LIN {X -0.212,Y -660.705,Z 1253.356,A 0.000,B 0.000,C 90.000,E1 100.141} C_DIS
LIN {X 0.232,Y -659.495,Z 1253.354,A 0.000,B 0.000,C 90.000,E1 99.613} C_DIS
LIN {X 0.124,Y -658.795,Z 1253.352,A 0.000,B 0.000,C 90.000,E1 99.378} C_DIS
LIN {X -0.205,Y -657.112,Z 1253.349,A 0.000,B 0.000,C 90.000,E1 98.916} C_DIS
LIN {X 0.108,Y -655.018,Z 1253.347,A 0.000,B 0.000,C 90.000,E1 98.398} C_DIS
LIN {X -0.260,Y -651.900,Z 1253.343,A 0.000,B 0.000,C 90.000,E1 97.814} C_DIS
LIN {X 0.015,Y -649.059,Z 1253.341,A 0.000,B 0.000,C 90.000,E1 97.296} C_DIS
LIN {X 0.153,Y -644.946,Z 1253.337,A 0.000,B 0.000,C 90.000,E1 96.663} C_DIS
LIN {X 0.258,Y -640.230,Z 1253.334,A 0.000,B 0.000,C 90.000,E1 96.030} C_DIS
LIN {X -0.052,Y -637.232,Z 1253.332,A 0.000,B 0.000,C 90.000,E1 95.682} C_DIS
LIN {X -0.011,Y -631.428,Z 1253.328,A 0.000,B 0.000,C 90.000,E1 95.049} C_DIS
LIN {X 0.272,Y -626.430,Z 1253.325,A 0.000,B 0.000,C 90.000,E1 94.531} C_DIS
LIN {X 0.030,Y -619.785,Z 1253.322,A 0.000,B 0.000,C 90.000,E1 93.955} C_DIS
LIN {X 0.104,Y -612.877,Z 1253.319,A 0.000,B 0.000,C 90.000,E1 93.383} C_DIS
LIN {X 0.178,Y -610.033,Z 1253.318,A 0.000,B 0.000,C 90.000,E1 93.154} C_DIS
LIN {X 0.140,Y -602.473,Z 1253.315,A 0.000,B 0.000,C 90.000,E1 92.636} C_DIS
LIN {X 0.166,Y -596.282,Z 1253.313,A 0.000,B 0.000,C 90.000,E1 92.236} C_DIS
LIN {X -0.229,Y -589.784,Z 1253.310,A 0.000,B 0.000,C 90.000,E1 91.892} C_DIS
LIN {X -0.265,Y -582.813,Z 1253.308,A 0.000,B 0.000,C 90.000,E1 91.547} C_DIS
LIN {X 0.065,Y -571.892,Z 1253.306,A 0.000,B 0.000,C 90.000,E1 91.088} C_DIS
LIN {X -0.005,Y -570.760,Z 1253.306,A 0.000,B 0.000,C 90.000,E1 91.031} C_DIS
LIN {X -0.074,Y -568.415,Z 1253.305,A 0.000,B 0.000,C 90.000,E1 90.859} C_DIS
LIN {X -0.108,Y -568.400,Z 1253.305,A 0.000,B 0.000,C 90.000,E1 90.859} C_DIS
LIN {X -0.110,Y -567.219,Z 1253.303,A 0.000,B 0.000,C 90.000,E1 90.516} C_DIS
LIN {X 0.015,Y -567.116,Z 1253.300,A 0.000,B 0.000,C 90.000,E1 90.057} C_DIS
LIN {X 0.207,Y -568.765,Z 1253.287,A 0.000,B 0.000,C 90.000,E1 87.707} C_DIS
LIN {X 0.001,Y -570.383,Z 1253.277,A 0.000,B 0.000,C 90.000,E1 85.812} C_DIS
LIN {X 0.269,Y -572.026,Z 1253.268,A 0.000,B 0.000,C 90.000,E1 84.147} C_DIS
LIN {X -0.071,Y -573.481,Z 1253.260,A 0.000,B 0.000,C 90.000,E1 82.818} C_DIS
LIN {X 0.021,Y -575.454,Z 1253.250,A 0.000,B 0.000,C 90.000,E1 80.905} C_DIS
LIN {X 0.191,Y -576.493,Z 1253.244,A 0.000,B 0.000,C 90.000,E1 79.803} C_DIS
LIN {X 0.012,Y -577.547,Z 1253.236,A 0.000,B 0.000,C 90.000,E1 78.465} C_DIS
LIN {X -0.254,Y -578.363,Z 1253.230,A 0.000,B 0.000,C 90.000,E1 77.409} C_DIS
LIN {X 0.065,Y -579.449,Z 1253.221,A 0.000,B 0.000,C 90.000,E1 75.755} C_DIS
LIN {X 0.188,Y -580.267,Z 1253.214,A 0.000,B 0.000,C 90.000,E1 74.393} C_DIS
LIN {X -0.241,Y -581.061,Z 1253.206,A 0.000,B 0.000,C 90.000,E1 73.087} C_DIS
LIN {X 0.106,Y -582.211,Z 1253.195,A 0.000,B 0.000,C 90.000,E1 71.167} C_DIS
LIN {X -0.144,Y -582.836,Z 1253.189,A 0.000,B 0.000,C 90.000,E1 70.115} C_DIS
LIN {X -0.251,Y -584.179,Z 1253.178,A 0.000,B 0.000,C 90.000,E1 67.975} C_DIS
LIN {X -0.130,Y -586.270,Z 1253.163,A 0.000,B 0.000,C 90.000,E1 65.281} C_DIS
LIN {X 0.004,Y -588.112,Z 1253.151,A 0.000,B 0.000,C 90.000,E1 63.127} C_DIS
LIN {X 0.091,Y -590.450,Z 1253.137,A 0.000,B 0.000,C 90.000,E1 60.717} C_DIS
LIN {X -0.152,Y -591.819,Z 1253.130,A 0.000,B 0.000,C 90.000,E1 59.410} C_DIS
LIN {X 0.030,Y -592.949,Z 1253.124,A 0.000,B 0.000,C 90.000,E1 58.329} C_DIS
LIN {X 0.120,Y -594.284,Z 1253.117,A 0.000,B 0.000,C 90.000,E1 56.993} C_DIS
LIN {X 0.277,Y -595.738,Z 1253.108,A 0.000,B 0.000,C 90.000,E1 55.388} C_DIS
LIN {X -0.244,Y -596.930,Z 1253.101,A 0.000,B 0.000,C 90.000,E1 54.116} C_DIS
LIN {X 0.326,Y -598.249,Z 1253.092,A 0.000,B 0.000,C 90.000,E1 52.477} C_DIS
LIN {X 0.204,Y -599.273,Z 1253.084,A 0.000,B 0.000,C 90.000,E1 51.170} C_DIS
LIN {X -0.149,Y -599.925,Z 1253.079,A 0.000,B 0.000,C 90.000,E1 50.150} C_DIS
LIN {X -0.307,Y -600.765,Z 1253.068,A 0.000,B 0.000,C 90.000,E1 48.324} C_DIS
LIN {X -0.064,Y -601.171,Z 1253.061,A 0.000,B 0.000,C 90.000,E1 46.986} C_DIS
LIN {X 0.188,Y -601.494,Z 1253.054,A 0.000,B 0.000,C 90.000,E1 45.648} C_DIS
LIN {X 0.217,Y -601.534,Z 1253.048,A 0.000,B 0.000,C 90.000,E1 44.595} C_DIS
LIN {X 0.244,Y -601.354,Z 1253.042,A 0.000,B 0.000,C 90.000,E1 43.542} C_DIS
LIN {X -0.148,Y -601.034,Z 1253.036,A 0.000,B 0.000,C 90.000,E1 42.528} C_DIS
LIN {X -0.069,Y -600.444,Z 1253.027,A 0.000,B 0.000,C 90.000,E1 40.943} C_DIS
LIN {X -0.019,Y -599.846,Z 1253.022,A 0.000,B 0.000,C 90.000,E1 39.886} C_DIS
LIN {X 0.258,Y -599.022,Z 1253.014,A 0.000,B 0.000,C 90.000,E1 38.543} C_DIS
LIN {X -0.334,Y -598.349,Z 1253.010,A 0.000,B 0.000,C 90.000,E1 37.810} C_DIS
LIN {X 0.136,Y -597.246,Z 1253.004,A 0.000,B 0.000,C 90.000,E1 36.710} C_DIS
LIN {X -0.119,Y -595.857,Z 1252.998,A 0.000,B 0.000,C 90.000,E1 35.678} C_DIS
LIN {X -0.149,Y -595.087,Z 1252.995,A 0.000,B 0.000,C 90.000,E1 35.152} C_DIS
LIN {X 0.064,Y -593.240,Z 1252.989,A 0.000,B 0.000,C 90.000,E1 34.072} C_DIS
LIN {X 0.090,Y -591.042,Z 1252.984,A 0.000,B 0.000,C 90.000,E1 33.007} C_DIS
LIN {X 0.056,Y -589.056,Z 1252.979,A 0.000,B 0.000,C 90.000,E1 32.212} C_DIS
LIN {X 0.010,Y -586.738,Z 1252.975,A 0.000,B 0.000,C 90.000,E1 31.416} C_DIS
LIN {X 0.243,Y -584.098,Z 1252.970,A 0.000,B 0.000,C 90.000,E1 30.590} C_DIS
LIN {X 0.143,Y -580.969,Z 1252.966,A 0.000,B 0.000,C 90.000,E1 29.795} C_DIS
LIN {X -0.130,Y -578.685,Z 1252.963,A 0.000,B 0.000,C 90.000,E1 29.283} C_DIS
LIN {X -0.133,Y -576.179,Z 1252.960,A 0.000,B 0.000,C 90.000,E1 28.743} C_DIS
LIN {X 0.069,Y -573.479,Z 1252.957,A 0.000,B 0.000,C 90.000,E1 28.180} C_DIS
LIN {X 0.019,Y -570.606,Z 1252.954,A 0.000,B 0.000,C 90.000,E1 27.641} C_DIS
LIN {X 0.100,Y -566.694,Z 1252.950,A 0.000,B 0.000,C 90.000,E1 26.950} C_DIS
LIN {X -0.007,Y -563.312,Z 1252.947,A 0.000,B 0.000,C 90.000,E1 26.411} C_DIS
LIN {X -0.088,Y -557.862,Z 1252.942,A 0.000,B 0.000,C 90.000,E1 25.591} C_DIS
LIN {X -0.112,Y -552.822,Z 1252.938,A 0.000,B 0.000,C 90.000,E1 24.899} C_DIS
LIN {X -0.222,Y -546.312,Z 1252.934,A 0.000,B 0.000,C 90.000,E1 24.079} C_DIS
LIN {X 0.149,Y -540.407,Z 1252.930,A 0.000,B 0.000,C 90.000,E1 23.334} C_DIS
LIN {X 0.178,Y -533.117,Z 1252.925,A 0.000,B 0.000,C 90.000,E1 22.514} C_DIS
LIN {X -0.235,Y -525.243,Z 1252.921,A 0.000,B 0.000,C 90.000,E1 21.716} C_DIS
LIN {X 0.015,Y -516.052,Z 1252.915,A 0.000,B 0.000,C 90.000,E1 20.737} C_DIS
LIN {X -0.065,Y -505.488,Z 1252.909,A 0.000,B 0.000,C 90.000,E1 19.685} C_DIS
LIN {X 0.052,Y -495.616,Z 1252.904,A 0.000,B 0.000,C 90.000,E1 18.725} C_DIS
LIN {X -0.104,Y -486.934,Z 1252.900,A 0.000,B 0.000,C 90.000,E1 17.946} C_DIS
LIN {X -0.065,Y -478.380,Z 1252.895,A 0.000,B 0.000,C 90.000,E1 17.166} C_DIS
LIN {X -0.049,Y -462.047,Z 1252.887,A 0.000,B 0.000,C 90.000,E1 15.717} C_DIS
LIN {X -0.194,Y -444.342,Z 1252.878,A 0.000,B 0.000,C 90.000,E1 14.120} C_DIS
LIN {X -0.038,Y -421.556,Z 1252.866,A 0.000,B 0.000,C 90.000,E1 11.827} C_DIS
LIN {X 0.078,Y -407.325,Z 1252.857,A 0.000,B 0.000,C 90.000,E1 10.254} C_DIS
LIN {X 0.105,Y -401.563,Z 1252.854,A 0.000,B 0.000,C 90.000,E1 9.613} C_DIS
LIN {X 0.063,Y -397.092,Z 1252.850,A 0.000,B 0.000,C 90.000,E1 9.029} C_DIS
LIN {X 0.041,Y -395.063,Z 1252.848,A 0.000,B 0.000,C 90.000,E1 8.681} C_DIS
LIN {X 0.176,Y -394.571,Z 1252.848,A 0.000,B 0.000,C 90.000,E1 8.568} C_DIS
LIN {X 0.138,Y -394.543,Z 1252.848,A 0.000,B 0.000,C 90.000,E1 8.568} C_DIS
LIN {X 0.073,Y -394.451,Z 1252.847,A 0.000,B 0.000,C 90.000,E1 8.511} C_DIS
LIN {X 0.035,Y -394.445,Z 1252.847,A 0.000,B 0.000,C 90.000,E1 8.511} C_DIS
LIN {X 0.137,Y -396.450,Z 1252.845,A 0.000,B 0.000,C 90.000,E1 8.049} C_DIS
LIN {X -0.191,Y -399.766,Z 1252.843,A 0.000,B 0.000,C 90.000,E1 7.757} C_DIS
LIN {X 0.059,Y -403.844,Z 1252.841,A 0.000,B 0.000,C 90.000,E1 7.409} C_DIS
LIN {X -0.125,Y -413.483,Z 1252.838,A 0.000,B 0.000,C 90.000,E1 6.777} C_DIS
LIN {X -0.006,Y -423.027,Z 1252.834,A 0.000,B 0.000,C 90.000,E1 6.087} C_DIS
LIN {X -0.107,Y -430.941,Z 1252.831,A 0.000,B 0.000,C 90.000,E1 5.511} C_DIS
LIN {X 0.128,Y -438.553,Z 1252.827,A 0.000,B 0.000,C 90.000,E1 4.878} C_DIS
LIN {X -0.106,Y -452.599,Z 1252.821,A 0.000,B 0.000,C 90.000,E1 3.784} C_DIS
LIN {X -0.122,Y -460.203,Z 1252.818,A 0.000,B 0.000,C 90.000,E1 3.154} C_DIS
LIN {X 0.232,Y -467.575,Z 1252.814,A 0.000,B 0.000,C 90.000,E1 2.465} C_DIS
LIN {X 0.122,Y -473.346,Z 1252.811,A 0.000,B 0.000,C 90.000,E1 1.949} C_DIS
LIN {X -0.172,Y -478.953,Z 1252.808,A 0.000,B 0.000,C 90.000,E1 1.432} C_DIS
LIN {X 0.010,Y -485.708,Z 1252.804,A 0.000,B 0.000,C 90.000,E1 0.688} C_DIS
LIN {X 0.000,Y -491.571,Z 1252.800,A 0.000,B 0.000,C 90.000,E1 360.000} C_DIS
LIN {X 0.034,Y -495.782,Z 1252.797,A 0.000,B 0.000,C 90.000,E1 359.484} C_DIS
LIN {X -0.059,Y -501.360,Z 1252.793,A 0.000,B 0.000,C 90.000,E1 358.740} C_DIS
LIN {X -0.089,Y -506.541,Z 1252.789,A 0.000,B 0.000,C 90.000,E1 357.993} C_DIS
LIN {X -0.087,Y -511.392,Z 1252.785,A 0.000,B 0.000,C 90.000,E1 357.249} C_DIS
LIN {X 0.202,Y -516.817,Z 1252.780,A 0.000,B 0.000,C 90.000,E1 356.331} C_DIS
LIN {X -0.129,Y -519.389,Z 1252.777,A 0.000,B 0.000,C 90.000,E1 355.927} C_DIS
LIN {X 0.022,Y -523.280,Z 1252.773,A 0.000,B 0.000,C 90.000,E1 355.179} C_DIS
LIN {X 0.207,Y -526.904,Z 1252.769,A 0.000,B 0.000,C 90.000,E1 354.432} C_DIS
LIN {X 0.180,Y -529.625,Z 1252.766,A 0.000,B 0.000,C 90.000,E1 353.856} C_DIS
LIN {X 0.171,Y -532.171,Z 1252.763,A 0.000,B 0.000,C 90.000,E1 353.280} C_DIS
LIN {X 0.221,Y -535.546,Z 1252.758,A 0.000,B 0.000,C 90.000,E1 352.413} C_DIS
LIN {X -0.229,Y -538.689,Z 1252.753,A 0.000,B 0.000,C 90.000,E1 351.602} C_DIS
LIN {X -0.114,Y -541.618,Z 1252.749,A 0.000,B 0.000,C 90.000,E1 350.735} C_DIS
LIN {X 0.122,Y -544.158,Z 1252.744,A 0.000,B 0.000,C 90.000,E1 349.859} C_DIS
LIN {X -0.155,Y -547.318,Z 1252.738,A 0.000,B 0.000,C 90.000,E1 348.757} C_DIS
LIN {X -0.287,Y -550.077,Z 1252.731,A 0.000,B 0.000,C 90.000,E1 347.645} C_DIS
LIN {X -0.140,Y -553.217,Z 1252.724,A 0.000,B 0.000,C 90.000,E1 346.228} C_DIS
LIN {X -0.320,Y -554.809,Z 1252.719,A 0.000,B 0.000,C 90.000,E1 345.408} C_DIS
LIN {X -0.221,Y -556.749,Z 1252.713,A 0.000,B 0.000,C 90.000,E1 344.283} C_DIS
LIN {X 0.060,Y -558.427,Z 1252.706,A 0.000,B 0.000,C 90.000,E1 343.142} C_DIS
LIN {X -0.163,Y -559.792,Z 1252.700,A 0.000,B 0.000,C 90.000,E1 342.054} C_DIS
LIN {X 0.167,Y -560.813,Z 1252.694,A 0.000,B 0.000,C 90.000,E1 340.913} C_DIS
LIN {X -0.026,Y -561.387,Z 1252.688,A 0.000,B 0.000,C 90.000,E1 339.826} C_DIS
LIN {X -0.336,Y -561.509,Z 1252.683,A 0.000,B 0.000,C 90.000,E1 339.028} C_DIS
LIN {X 0.085,Y -561.263,Z 1252.679,A 0.000,B 0.000,C 90.000,E1 338.156} C_DIS
LIN {X -0.224,Y -560.706,Z 1252.674,A 0.000,B 0.000,C 90.000,E1 337.358} C_DIS
LIN {X 0.192,Y -559.841,Z 1252.670,A 0.000,B 0.000,C 90.000,E1 336.485} C_DIS
LIN {X 0.087,Y -558.671,Z 1252.665,A 0.000,B 0.000,C 90.000,E1 335.665} C_DIS
LIN {X -0.029,Y -557.185,Z 1252.660,A 0.000,B 0.000,C 90.000,E1 334.845} C_DIS
LIN {X 0.122,Y -554.796,Z 1252.654,A 0.000,B 0.000,C 90.000,E1 333.717} C_DIS
LIN {X -0.095,Y -554.002,Z 1252.653,A 0.000,B 0.000,C 90.000,E1 333.461} C_DIS
LIN {X -0.065,Y -553.388,Z 1252.651,A 0.000,B 0.000,C 90.000,E1 333.179} C_DIS
LIN {X -0.243,Y -550.785,Z 1252.646,A 0.000,B 0.000,C 90.000,E1 332.359} C_DIS
LIN {X -0.195,Y -547.731,Z 1252.642,A 0.000,B 0.000,C 90.000,E1 331.513} C_DIS
LIN {X 0.187,Y -546.009,Z 1252.639,A 0.000,B 0.000,C 90.000,E1 331.051} C_DIS
LIN {X -0.169,Y -542.745,Z 1252.635,A 0.000,B 0.000,C 90.000,E1 330.383} C_DIS
LIN {X -0.082,Y -539.018,Z 1252.631,A 0.000,B 0.000,C 90.000,E1 329.665} C_DIS
LIN {X 0.106,Y -535.654,Z 1252.628,A 0.000,B 0.000,C 90.000,E1 329.076} C_DIS
LIN {X 0.221,Y -528.187,Z 1252.622,A 0.000,B 0.000,C 90.000,E1 327.916} C_DIS
LIN {X 0.040,Y -520.383,Z 1252.616,A 0.000,B 0.000,C 90.000,E1 326.786} C_DIS
LIN {X 0.033,Y -515.805,Z 1252.612,A 0.000,B 0.000,C 90.000,E1 326.087} C_DIS
LIN {X -0.050,Y -512.575,Z 1252.609,A 0.000,B 0.000,C 90.000,E1 325.548} C_DIS
LIN {X -0.109,Y -509.785,Z 1252.606,A 0.000,B 0.000,C 90.000,E1 325.022} C_DIS
LIN {X 0.129,Y -507.435,Z 1252.602,A 0.000,B 0.000,C 90.000,E1 324.402} C_DIS
LIN {X -0.024,Y -505.761,Z 1252.599,A 0.000,B 0.000,C 90.000,E1 323.829} C_DIS
LIN {X 0.180,Y -504.597,Z 1252.596,A 0.000,B 0.000,C 90.000,E1 323.210} C_DIS
LIN {X -0.034,Y -503.754,Z 1252.592,A 0.000,B 0.000,C 90.000,E1 322.637} C_DIS
LIN {X -0.056,Y -503.268,Z 1252.588,A 0.000,B 0.000,C 90.000,E1 321.743} C_DIS
LIN {X -0.012,Y -503.780,Z 1252.569,A 0.000,B 0.000,C 90.000,E1 318.447} C_DIS
LIN {X -0.210,Y -504.378,Z 1252.558,A 0.000,B 0.000,C 90.000,E1 316.377} C_DIS
LIN {X 0.195,Y -504.702,Z 1252.549,A 0.000,B 0.000,C 90.000,E1 314.838} C_DIS
LIN {X -0.109,Y -505.060,Z 1252.541,A 0.000,B 0.000,C 90.000,E1 313.380} C_DIS
LIN {X 0.057,Y -505.627,Z 1252.529,A 0.000,B 0.000,C 90.000,E1 311.272} C_DIS
LIN {X 0.060,Y -505.992,Z 1252.519,A 0.000,B 0.000,C 90.000,E1 309.483} C_DIS
LIN {X 0.056,Y -506.474,Z 1252.508,A 0.000,B 0.000,C 90.000,E1 307.397} C_DIS
LIN {X -0.040,Y -506.824,Z 1252.501,A 0.000,B 0.000,C 90.000,E1 306.217} C_DIS
LIN {X -0.029,Y -507.013,Z 1252.495,A 0.000,B 0.000,C 90.000,E1 305.025} C_DIS
LIN {X 0.302,Y -507.136,Z 1252.486,A 0.000,B 0.000,C 90.000,E1 303.499} C_DIS
LIN {X -0.018,Y -507.187,Z 1252.476,A 0.000,B 0.000,C 90.000,E1 301.750} C_DIS
LIN {X 0.149,Y -507.117,Z 1252.470,A 0.000,B 0.000,C 90.000,E1 300.541} C_DIS
LIN {X 0.261,Y -507.099,Z 1252.460,A 0.000,B 0.000,C 90.000,E1 298.743} C_DIS
LIN {X -0.122,Y -506.892,Z 1252.450,A 0.000,B 0.000,C 90.000,E1 297.001} C_DIS
LIN {X 0.127,Y -506.793,Z 1252.437,A 0.000,B 0.000,C 90.000,E1 294.591} C_DIS
LIN {X 0.246,Y -506.796,Z 1252.430,A 0.000,B 0.000,C 90.000,E1 293.387} C_DIS
LIN {X 0.253,Y -506.480,Z 1252.422,A 0.000,B 0.000,C 90.000,E1 291.897} C_DIS
LIN {X 0.158,Y -505.684,Z 1252.412,A 0.000,B 0.000,C 90.000,E1 290.120} C_DIS
LIN {X -0.113,Y -504.623,Z 1252.399,A 0.000,B 0.000,C 90.000,E1 287.764} C_DIS
LIN {X 0.051,Y -504.205,Z 1252.392,A 0.000,B 0.000,C 90.000,E1 286.551} C_DIS
LIN {X -0.014,Y -503.519,Z 1252.384,A 0.000,B 0.000,C 90.000,E1 285.064} C_DIS
LIN {X -0.217,Y -502.611,Z 1252.375,A 0.000,B 0.000,C 90.000,E1 283.592} C_DIS
LIN {X 0.054,Y -501.572,Z 1252.367,A 0.000,B 0.000,C 90.000,E1 282.063} C_DIS
LIN {X 0.202,Y -500.426,Z 1252.359,A 0.000,B 0.000,C 90.000,E1 280.546} C_DIS
LIN {X 0.170,Y -499.181,Z 1252.349,A 0.000,B 0.000,C 90.000,E1 278.746} C_DIS
LIN {X 0.103,Y -498.052,Z 1252.339,A 0.000,B 0.000,C 90.000,E1 276.947} C_DIS
LIN {X 0.138,Y -496.782,Z 1252.325,A 0.000,B 0.000,C 90.000,E1 274.531} C_DIS
LIN {X 0.106,Y -496.101,Z 1252.319,A 0.000,B 0.000,C 90.000,E1 273.326} C_DIS
LIN {X -0.070,Y -495.051,Z 1252.310,A 0.000,B 0.000,C 90.000,E1 271.835} C_DIS
LIN {X -0.210,Y -493.235,Z 1252.297,A 0.000,B 0.000,C 90.000,E1 269.427} C_DIS
LIN {X -0.046,Y -491.472,Z 1252.281,A 0.000,B 0.000,C 90.000,E1 266.674} C_DIS
LIN {X 0.048,Y -490.478,Z 1252.271,A 0.000,B 0.000,C 90.000,E1 264.837} C_DIS
LIN {X -0.161,Y -489.520,Z 1252.263,A 0.000,B 0.000,C 90.000,E1 263.337} C_DIS
LIN {X -0.269,Y -488.598,Z 1252.256,A 0.000,B 0.000,C 90.000,E1 262.129} C_DIS
LIN {X 0.108,Y -487.122,Z 1252.248,A 0.000,B 0.000,C 90.000,E1 260.557} C_DIS
LIN {X -0.027,Y -484.754,Z 1252.232,A 0.000,B 0.000,C 90.000,E1 257.813} C_DIS
LIN {X -0.086,Y -483.773,Z 1252.224,A 0.000,B 0.000,C 90.000,E1 256.284} C_DIS
LIN {X 0.128,Y -482.296,Z 1252.210,A 0.000,B 0.000,C 90.000,E1 253.795} C_DIS
LIN {X 0.108,Y -481.096,Z 1252.198,A 0.000,B 0.000,C 90.000,E1 251.638} C_DIS
LIN {X -0.083,Y -480.146,Z 1252.188,A 0.000,B 0.000,C 90.000,E1 249.806} C_DIS
LIN {X 0.158,Y -479.290,Z 1252.179,A 0.000,B 0.000,C 90.000,E1 248.230} C_DIS
LIN {X 0.275,Y -478.309,Z 1252.169,A 0.000,B 0.000,C 90.000,E1 246.357} C_DIS
LIN {X -0.046,Y -477.192,Z 1252.160,A 0.000,B 0.000,C 90.000,E1 244.845} C_DIS
LIN {X 0.063,Y -476.372,Z 1252.153,A 0.000,B 0.000,C 90.000,E1 243.589} C_DIS
LIN {X 0.127,Y -475.332,Z 1252.145,A 0.000,B 0.000,C 90.000,E1 242.025} C_DIS
LIN {X 0.175,Y -474.196,Z 1252.136,A 0.000,B 0.000,C 90.000,E1 240.461} C_DIS
LIN {X 0.028,Y -472.895,Z 1252.127,A 0.000,B 0.000,C 90.000,E1 238.918} C_DIS
LIN {X 0.030,Y -471.234,Z 1252.117,A 0.000,B 0.000,C 90.000,E1 237.041} C_DIS
LIN {X 0.004,Y -469.467,Z 1252.105,A 0.000,B 0.000,C 90.000,E1 234.848} C_DIS
LIN {X -0.093,Y -467.634,Z 1252.089,A 0.000,B 0.000,C 90.000,E1 232.029} C_DIS
LIN {X 0.047,Y -466.757,Z 1252.080,A 0.000,B 0.000,C 90.000,E1 230.436} C_DIS
LIN {X 0.102,Y -465.962,Z 1252.072,A 0.000,B 0.000,C 90.000,E1 228.852} C_DIS
LIN {X -0.208,Y -464.988,Z 1252.063,A 0.000,B 0.000,C 90.000,E1 227.310} C_DIS
LIN {X -0.019,Y -464.409,Z 1252.057,A 0.000,B 0.000,C 90.000,E1 226.338} C_DIS
LIN {X 0.075,Y -463.196,Z 1252.045,A 0.000,B 0.000,C 90.000,E1 224.109} C_DIS
LIN {X 0.105,Y -463.920,Z 1252.001,A 0.000,B 0.000,C 90.000,E1 216.171} C_DIS
LIN {X -0.204,Y -467.553,Z 1251.975,A 0.000,B 0.000,C 90.000,E1 211.465} C_DIS
LIN {X -0.065,Y -469.195,Z 1251.966,A 0.000,B 0.000,C 90.000,E1 209.873} C_DIS
LIN {X 0.047,Y -471.564,Z 1251.955,A 0.000,B 0.000,C 90.000,E1 207.975} C_DIS
LIN {X 0.120,Y -474.587,Z 1251.942,A 0.000,B 0.000,C 90.000,E1 205.463} C_DIS
LIN {X 0.153,Y -477.199,Z 1251.931,A 0.000,B 0.000,C 90.000,E1 203.590} C_DIS
LIN {X -0.192,Y -480.139,Z 1251.921,A 0.000,B 0.000,C 90.000,E1 201.770} C_DIS
LIN {X -0.198,Y -487.630,Z 1251.899,A 0.000,B 0.000,C 90.000,E1 197.764} C_DIS
LIN {X -0.032,Y -492.178,Z 1251.887,A 0.000,B 0.000,C 90.000,E1 195.607} C_DIS
LIN {X 0.086,Y -496.168,Z 1251.877,A 0.000,B 0.000,C 90.000,E1 193.772} C_DIS
LIN {X 0.104,Y -500.904,Z 1251.865,A 0.000,B 0.000,C 90.000,E1 191.658} C_DIS
LIN {X 0.205,Y -505.202,Z 1251.855,A 0.000,B 0.000,C 90.000,E1 189.849} C_DIS
LIN {X -0.142,Y -508.773,Z 1251.847,A 0.000,B 0.000,C 90.000,E1 188.398} C_DIS
LIN {X 0.073,Y -512.473,Z 1251.838,A 0.000,B 0.000,C 90.000,E1 186.891} C_DIS
LIN {X 0.208,Y -516.783,Z 1251.828,A 0.000,B 0.000,C 90.000,E1 185.106} C_DIS
LIN {X -0.118,Y -521.062,Z 1251.819,A 0.000,B 0.000,C 90.000,E1 183.383} C_DIS
LIN {X -0.248,Y -523.131,Z 1251.814,A 0.000,B 0.000,C 90.000,E1 182.522} C_DIS
LIN {X 0.058,Y -527.258,Z 1251.804,A 0.000,B 0.000,C 90.000,E1 180.745} C_DIS
LIN {X -0.097,Y -531.938,Z 1251.793,A 0.000,B 0.000,C 90.000,E1 178.740} C_DIS
LIN {X -0.127,Y -535.076,Z 1251.785,A 0.000,B 0.000,C 90.000,E1 177.306} C_DIS
LIN {X -0.105,Y -537.453,Z 1251.779,A 0.000,B 0.000,C 90.000,E1 176.159} C_DIS
LIN {X -0.010,Y -539.672,Z 1251.772,A 0.000,B 0.000,C 90.000,E1 175.008} C_DIS
LIN {X 0.125,Y -541.805,Z 1251.766,A 0.000,B 0.000,C 90.000,E1 173.856} C_DIS
LIN {X -0.173,Y -544.326,Z 1251.758,A 0.000,B 0.000,C 90.000,E1 172.470} C_DIS
LIN {X 0.107,Y -546.651,Z 1251.750,A 0.000,B 0.000,C 90.000,E1 171.027} C_DIS
LIN {X -0.143,Y -547.931,Z 1251.746,A 0.000,B 0.000,C 90.000,E1 170.208} C_DIS
LIN {X -0.150,Y -550.380,Z 1251.736,A 0.000,B 0.000,C 90.000,E1 168.522} C_DIS
LIN {X -0.125,Y -552.219,Z 1251.728,A 0.000,B 0.000,C 90.000,E1 167.117} C_DIS
LIN {X -0.240,Y -554.690,Z 1251.718,A 0.000,B 0.000,C 90.000,E1 165.172} C_DIS
LIN {X 0.127,Y -557.921,Z 1251.705,A 0.000,B 0.000,C 90.000,E1 162.906} C_DIS
LIN {X 0.201,Y -560.782,Z 1251.697,A 0.000,B 0.000,C 90.000,E1 161.511} C_DIS
LIN {X 0.146,Y -564.530,Z 1251.690,A 0.000,B 0.000,C 90.000,E1 160.134} C_DIS
LIN {X -0.134,Y -567.235,Z 1251.685,A 0.000,B 0.000,C 90.000,E1 159.337} C_DIS
LIN {X 0.226,Y -573.289,Z 1251.677,A 0.000,B 0.000,C 90.000,E1 157.794} C_DIS
LIN {X -0.268,Y -579.586,Z 1251.669,A 0.000,B 0.000,C 90.000,E1 156.485} C_DIS
LIN {X -0.116,Y -589.402,Z 1251.659,A 0.000,B 0.000,C 90.000,E1 154.588} C_DIS
LIN {X -0.042,Y -595.848,Z 1251.652,A 0.000,B 0.000,C 90.000,E1 153.384} C_DIS
LIN {X 0.125,Y -602.111,Z 1251.646,A 0.000,B 0.000,C 90.000,E1 152.180} C_DIS
LIN {X 0.158,Y -607.430,Z 1251.640,A 0.000,B 0.000,C 90.000,E1 151.129} C_DIS
LIN {X -0.284,Y -613.138,Z 1251.633,A 0.000,B 0.000,C 90.000,E1 149.999} C_DIS
LIN {X -0.100,Y -618.079,Z 1251.627,A 0.000,B 0.000,C 90.000,E1 148.948} C_DIS
LIN {X -0.057,Y -622.984,Z 1251.622,A 0.000,B 0.000,C 90.000,E1 147.916} C_DIS
LIN {X 0.251,Y -626.523,Z 1251.618,A 0.000,B 0.000,C 90.000,E1 147.120} C_DIS
LIN {X -0.112,Y -630.963,Z 1251.612,A 0.000,B 0.000,C 90.000,E1 146.135} C_DIS
LIN {X 0.112,Y -635.093,Z 1251.606,A 0.000,B 0.000,C 90.000,E1 145.102} C_DIS
LIN {X -0.133,Y -638.991,Z 1251.601,A 0.000,B 0.000,C 90.000,E1 144.116} C_DIS
LIN {X -0.331,Y -642.466,Z 1251.595,A 0.000,B 0.000,C 90.000,E1 143.130} C_DIS
LIN {X -0.005,Y -644.870,Z 1251.591,A 0.000,B 0.000,C 90.000,E1 142.351} C_DIS
LIN {X -0.164,Y -647.119,Z 1251.587,A 0.000,B 0.000,C 90.000,E1 141.618} C_DIS
LIN {X 0.128,Y -649.963,Z 1251.581,A 0.000,B 0.000,C 90.000,E1 140.598} C_DIS
LIN {X -0.044,Y -652.657,Z 1251.576,A 0.000,B 0.000,C 90.000,E1 139.622} C_DIS
LIN {X -0.228,Y -655.941,Z 1251.569,A 0.000,B 0.000,C 90.000,E1 138.405} C_DIS
LIN {X 0.084,Y -659.085,Z 1251.562,A 0.000,B 0.000,C 90.000,E1 137.148} C_DIS
LIN {X -0.066,Y -664.648,Z 1251.550,A 0.000,B 0.000,C 90.000,E1 134.960} C_DIS
LIN {X -0.064,Y -669.295,Z 1251.540,A 0.000,B 0.000,C 90.000,E1 133.257} C_DIS
LIN {X -0.454,Y -673.284,Z 1251.532,A 0.000,B 0.000,C 90.000,E1 131.838} C_DIS
LIN {X -0.299,Y -676.540,Z 1251.526,A 0.000,B 0.000,C 90.000,E1 130.620} C_DIS
LIN {X 0.027,Y -680.306,Z 1251.518,A 0.000,B 0.000,C 90.000,E1 129.152} C_DIS
LIN {X -0.135,Y -683.438,Z 1251.511,A 0.000,B 0.000,C 90.000,E1 127.971} C_DIS
LIN {X 0.324,Y -687.147,Z 1251.503,A 0.000,B 0.000,C 90.000,E1 126.503} C_DIS
LIN {X -0.200,Y -689.408,Z 1251.498,A 0.000,B 0.000,C 90.000,E1 125.598} C_DIS
LIN {X -0.091,Y -692.088,Z 1251.491,A 0.000,B 0.000,C 90.000,E1 124.405} C_DIS
LIN {X 0.024,Y -694.104,Z 1251.486,A 0.000,B 0.000,C 90.000,E1 123.452} C_DIS
LIN {X -0.153,Y -696.980,Z 1251.478,A 0.000,B 0.000,C 90.000,E1 122.054} C_DIS
LIN {X -0.091,Y -699.143,Z 1251.472,A 0.000,B 0.000,C 90.000,E1 120.875} C_DIS
LIN {X 0.373,Y -701.187,Z 1251.465,A 0.000,B 0.000,C 90.000,E1 119.667} C_DIS
LIN {X 0.238,Y -702.592,Z 1251.460,A 0.000,B 0.000,C 90.000,E1 118.743} C_DIS
LIN {X -0.214,Y -703.742,Z 1251.455,A 0.000,B 0.000,C 90.000,E1 117.847} C_DIS
LIN {X 0.302,Y -704.627,Z 1251.449,A 0.000,B 0.000,C 90.000,E1 116.873} C_DIS
LIN {X 0.222,Y -704.991,Z 1251.446,A 0.000,B 0.000,C 90.000,E1 116.181} C_DIS
LIN {X 0.167,Y -705.110,Z 1251.443,A 0.000,B 0.000,C 90.000,E1 115.720} C_DIS
LIN {X 0.093,Y -704.864,Z 1251.439,A 0.000,B 0.000,C 90.000,E1 115.027} C_DIS
LIN {X -0.265,Y -704.481,Z 1251.437,A 0.000,B 0.000,C 90.000,E1 114.591} C_DIS
LIN {X 0.305,Y -703.686,Z 1251.434,A 0.000,B 0.000,C 90.000,E1 114.079} C_DIS
LIN {X -0.341,Y -703.002,Z 1251.433,A 0.000,B 0.000,C 90.000,E1 113.898} C_DIS
LIN {X 0.217,Y -700.978,Z 1251.430,A 0.000,B 0.000,C 90.000,E1 113.387} C_DIS
LIN {X 0.353,Y -700.259,Z 1251.429,A 0.000,B 0.000,C 90.000,E1 113.259} C_DIS
LIN {X -0.035,Y -696.034,Z 1251.427,A 0.000,B 0.000,C 90.000,E1 112.823} C_DIS
LIN {X 0.093,Y -694.744,Z 1251.426,A 0.000,B 0.000,C 90.000,E1 112.695} C_DIS
LIN {X 0.010,Y -692.786,Z 1251.426,A 0.000,B 0.000,C 90.000,E1 112.589} C_DIS
LIN {X 0.094,Y -687.962,Z 1251.425,A 0.000,B 0.000,C 90.000,E1 112.408} C_DIS
LIN {X 0.256,Y -685.952,Z 1251.424,A 0.000,B 0.000,C 90.000,E1 112.333} C_DIS
LIN {X -0.193,Y -677.441,Z 1251.424,A 0.000,B 0.000,C 90.000,E1 112.259} C_DIS
LIN {X 0.393,Y -676.916,Z 1251.424,A 0.000,B 0.000,C 90.000,E1 112.206} C_DIS
LIN {X 0.327,Y -627.513,Z 1251.424,A 0.000,B 0.000,C 90.000,E1 112.206} C_DIS
LIN {X -0.031,Y -626.466,Z 1251.423,A 0.000,B 0.000,C 90.000,E1 112.206} C_DIS
LIN {X -0.088,Y -625.366,Z 1251.423,A 0.000,B 0.000,C 90.000,E1 112.153} C_DIS
LIN {X -0.240,Y -623.489,Z 1251.422,A 0.000,B 0.000,C 90.000,E1 112.025} C_DIS
LIN {X -0.276,Y -623.476,Z 1251.422,A 0.000,B 0.000,C 90.000,E1 112.025} C_DIS
LIN {X -0.104,Y -623.241,Z 1251.422,A 0.000,B 0.000,C 90.000,E1 111.897} C_DIS
LIN {X 0.096,Y -624.519,Z 1251.419,A 0.000,B 0.000,C 90.000,E1 111.482} C_DIS
LIN {X 0.092,Y -627.194,Z 1251.417,A 0.000,B 0.000,C 90.000,E1 110.972} C_DIS
LIN {X -0.076,Y -632.344,Z 1251.412,A 0.000,B 0.000,C 90.000,E1 110.120} C_DIS
LIN {X -0.374,Y -636.282,Z 1251.408,A 0.000,B 0.000,C 90.000,E1 109.396} C_DIS
LIN {X -0.241,Y -642.292,Z 1251.401,A 0.000,B 0.000,C 90.000,E1 108.127} C_DIS
LIN {X -0.151,Y -649.418,Z 1251.392,A 0.000,B 0.000,C 90.000,E1 106.622} C_DIS
LIN {X 0.253,Y -652.682,Z 1251.388,A 0.000,B 0.000,C 90.000,E1 105.843} C_DIS
LIN {X 0.004,Y -654.638,Z 1251.385,A 0.000,B 0.000,C 90.000,E1 105.371} C_DIS
LIN {X -0.179,Y -657.121,Z 1251.381,A 0.000,B 0.000,C 90.000,E1 104.647} C_DIS
LIN {X 0.237,Y -658.503,Z 1251.379,A 0.000,B 0.000,C 90.000,E1 104.120} C_DIS
LIN {X -0.078,Y -659.996,Z 1251.375,A 0.000,B 0.000,C 90.000,E1 103.411} C_DIS
LIN {X 0.362,Y -660.734,Z 1251.372,A 0.000,B 0.000,C 90.000,E1 102.883} C_DIS
LIN {X 0.164,Y -661.217,Z 1251.369,A 0.000,B 0.000,C 90.000,E1 102.411} C_DIS
LIN {X -0.171,Y -661.335,Z 1251.366,A 0.000,B 0.000,C 90.000,E1 101.951} C_DIS
LIN {X -0.267,Y -661.311,Z 1251.365,A 0.000,B 0.000,C 90.000,E1 101.715} C_DIS
LIN {X 0.185,Y -660.980,Z 1251.362,A 0.000,B 0.000,C 90.000,E1 101.186} C_DIS
LIN {X -0.016,Y -660.411,Z 1251.360,A 0.000,B 0.000,C 90.000,E1 100.715} C_DIS
LIN {X 0.307,Y -659.531,Z 1251.357,A 0.000,B 0.000,C 90.000,E1 100.197} C_DIS
LIN {X 0.092,Y -658.371,Z 1251.354,A 0.000,B 0.000,C 90.000,E1 99.726} C_DIS
LIN {X -0.129,Y -657.735,Z 1251.353,A 0.000,B 0.000,C 90.000,E1 99.500} C_DIS
LIN {X 0.289,Y -656.043,Z 1251.350,A 0.000,B 0.000,C 90.000,E1 98.973} C_DIS
LIN {X -0.054,Y -653.991,Z 1251.347,A 0.000,B 0.000,C 90.000,E1 98.511} C_DIS
LIN {X 0.214,Y -650.930,Z 1251.344,A 0.000,B 0.000,C 90.000,E1 97.871} C_DIS
LIN {X -0.279,Y -647.352,Z 1251.340,A 0.000,B 0.000,C 90.000,E1 97.296} C_DIS
LIN {X -0.034,Y -644.064,Z 1251.338,A 0.000,B 0.000,C 90.000,E1 96.777} C_DIS
LIN {X 0.063,Y -639.397,Z 1251.334,A 0.000,B 0.000,C 90.000,E1 96.144} C_DIS
LIN {X 0.297,Y -635.316,Z 1251.331,A 0.000,B 0.000,C 90.000,E1 95.625} C_DIS
LIN {X -0.130,Y -630.685,Z 1251.329,A 0.000,B 0.000,C 90.000,E1 95.163} C_DIS
LIN {X 0.163,Y -624.448,Z 1251.325,A 0.000,B 0.000,C 90.000,E1 94.531} C_DIS
LIN {X -0.067,Y -617.714,Z 1251.322,A 0.000,B 0.000,C 90.000,E1 93.955} C_DIS
LIN {X -0.020,Y -610.651,Z 1251.319,A 0.000,B 0.000,C 90.000,E1 93.383} C_DIS
LIN {X -0.239,Y -604.655,Z 1251.317,A 0.000,B 0.000,C 90.000,E1 92.980} C_DIS
LIN {X -0.082,Y -597.007,Z 1251.314,A 0.000,B 0.000,C 90.000,E1 92.465} C_DIS
LIN {X -0.261,Y -588.955,Z 1251.311,A 0.000,B 0.000,C 90.000,E1 92.007} C_DIS
LIN {X -0.247,Y -581.992,Z 1251.309,A 0.000,B 0.000,C 90.000,E1 91.661} C_DIS
LIN {X 0.166,Y -571.236,Z 1251.307,A 0.000,B 0.000,C 90.000,E1 91.203} C_DIS
LIN {X 0.062,Y -570.056,Z 1251.306,A 0.000,B 0.000,C 90.000,E1 91.146} C_DIS
LIN {X 0.167,Y -567.933,Z 1251.306,A 0.000,B 0.000,C 90.000,E1 90.974} C_DIS
LIN {X 0.132,Y -567.903,Z 1251.306,A 0.000,B 0.000,C 90.000,E1 90.974} C_DIS
LIN {X 0.030,Y -567.764,Z 1251.305,A 0.000,B 0.000,C 90.000,E1 90.859} C_DIS
LIN {X 0.041,Y -566.945,Z 1251.303,A 0.000,B 0.000,C 90.000,E1 90.516} C_DIS
LIN {X -0.174,Y -567.007,Z 1251.300,A 0.000,B 0.000,C 90.000,E1 90.057} C_DIS
LIN {X -0.024,Y -568.202,Z 1251.291,A 0.000,B 0.000,C 90.000,E1 88.396} C_DIS
LIN {X -0.254,Y -569.747,Z 1251.281,A 0.000,B 0.000,C 90.000,E1 86.502} C_DIS
LIN {X -0.271,Y -571.840,Z 1251.268,A 0.000,B 0.000,C 90.000,E1 84.318} C_DIS
LIN {X -0.042,Y -573.280,Z 1251.261,A 0.000,B 0.000,C 90.000,E1 82.932} C_DIS
LIN {X -0.040,Y -575.238,Z 1251.250,A 0.000,B 0.000,C 90.000,E1 81.027} C_DIS
LIN {X 0.118,Y -576.264,Z 1251.244,A 0.000,B 0.000,C 90.000,E1 79.926} C_DIS
LIN {X -0.171,Y -577.147,Z 1251.238,A 0.000,B 0.000,C 90.000,E1 78.870} C_DIS
LIN {X -0.222,Y -578.131,Z 1251.231,A 0.000,B 0.000,C 90.000,E1 77.521} C_DIS
LIN {X 0.086,Y -578.878,Z 1251.225,A 0.000,B 0.000,C 90.000,E1 76.408} C_DIS
LIN {X 0.197,Y -579.754,Z 1251.217,A 0.000,B 0.000,C 90.000,E1 75.046} C_DIS
LIN {X -0.023,Y -580.706,Z 1251.208,A 0.000,B 0.000,C 90.000,E1 73.449} C_DIS
LIN {X -0.237,Y -581.782,Z 1251.198,A 0.000,B 0.000,C 90.000,E1 71.583} C_DIS
LIN {X 0.260,Y -582.606,Z 1251.190,A 0.000,B 0.000,C 90.000,E1 70.188} C_DIS
LIN {X 0.135,Y -583.951,Z 1251.178,A 0.000,B 0.000,C 90.000,E1 68.050} C_DIS
LIN {X 0.235,Y -586.038,Z 1251.163,A 0.000,B 0.000,C 90.000,E1 65.357} C_DIS
LIN {X -0.172,Y -587.877,Z 1251.151,A 0.000,B 0.000,C 90.000,E1 63.256} C_DIS
LIN {X -0.091,Y -590.208,Z 1251.138,A 0.000,B 0.000,C 90.000,E1 60.845} C_DIS
LIN {X -0.337,Y -591.576,Z 1251.131,A 0.000,B 0.000,C 90.000,E1 59.537} C_DIS
LIN {X -0.265,Y -592.982,Z 1251.123,A 0.000,B 0.000,C 90.000,E1 58.201} C_DIS
LIN {X -0.068,Y -594.078,Z 1251.117,A 0.000,B 0.000,C 90.000,E1 57.120} C_DIS
LIN {X 0.088,Y -595.499,Z 1251.109,A 0.000,B 0.000,C 90.000,E1 55.515} C_DIS
LIN {X 0.051,Y -596.704,Z 1251.101,A 0.000,B 0.000,C 90.000,E1 54.196} C_DIS
LIN {X 0.010,Y -598.247,Z 1251.091,A 0.000,B 0.000,C 90.000,E1 52.351} C_DIS
LIN {X 0.018,Y -599.047,Z 1251.085,A 0.000,B 0.000,C 90.000,E1 51.295} C_DIS
LIN {X 0.128,Y -599.725,Z 1251.079,A 0.000,B 0.000,C 90.000,E1 50.231} C_DIS
LIN {X -0.056,Y -600.299,Z 1251.072,A 0.000,B 0.000,C 90.000,E1 48.933} C_DIS
LIN {X -0.248,Y -600.634,Z 1251.068,A 0.000,B 0.000,C 90.000,E1 48.162} C_DIS
LIN {X 0.411,Y -600.974,Z 1251.063,A 0.000,B 0.000,C 90.000,E1 47.310} C_DIS
LIN {X 0.031,Y -601.273,Z 1251.054,A 0.000,B 0.000,C 90.000,E1 45.769} C_DIS
LIN {X 0.050,Y -601.384,Z 1251.048,A 0.000,B 0.000,C 90.000,E1 44.717} C_DIS
LIN {X -0.348,Y -601.210,Z 1251.043,A 0.000,B 0.000,C 90.000,E1 43.704} C_DIS
LIN {X 0.317,Y -600.990,Z 1251.038,A 0.000,B 0.000,C 90.000,E1 42.852} C_DIS
LIN {X -0.290,Y -600.520,Z 1251.031,A 0.000,B 0.000,C 90.000,E1 41.595} C_DIS
LIN {X -0.245,Y -600.031,Z 1251.025,A 0.000,B 0.000,C 90.000,E1 40.539} C_DIS
LIN {X 0.014,Y -599.562,Z 1251.021,A 0.000,B 0.000,C 90.000,E1 39.725} C_DIS
LIN {X 0.044,Y -598.938,Z 1251.015,A 0.000,B 0.000,C 90.000,E1 38.669} C_DIS
LIN {X -0.081,Y -598.280,Z 1251.010,A 0.000,B 0.000,C 90.000,E1 37.890} C_DIS
LIN {X -0.211,Y -596.862,Z 1251.003,A 0.000,B 0.000,C 90.000,E1 36.583} C_DIS
LIN {X -0.120,Y -595.421,Z 1250.997,A 0.000,B 0.000,C 90.000,E1 35.518} C_DIS
LIN {X -0.011,Y -594.591,Z 1250.994,A 0.000,B 0.000,C 90.000,E1 34.978} C_DIS
LIN {X 0.044,Y -592.719,Z 1250.989,A 0.000,B 0.000,C 90.000,E1 33.913} C_DIS
LIN {X -0.265,Y -590.415,Z 1250.983,A 0.000,B 0.000,C 90.000,E1 32.880} C_DIS
LIN {X -0.182,Y -589.100,Z 1250.980,A 0.000,B 0.000,C 90.000,E1 32.339} C_DIS
LIN {X -0.109,Y -587.619,Z 1250.977,A 0.000,B 0.000,C 90.000,E1 31.799} C_DIS
LIN {X -0.170,Y -585.090,Z 1250.972,A 0.000,B 0.000,C 90.000,E1 31.003} C_DIS
LIN {X 0.004,Y -584.225,Z 1250.971,A 0.000,B 0.000,C 90.000,E1 30.718} C_DIS
LIN {X -0.094,Y -581.114,Z 1250.966,A 0.000,B 0.000,C 90.000,E1 29.922} C_DIS
LIN {X 0.281,Y -577.676,Z 1250.962,A 0.000,B 0.000,C 90.000,E1 29.077} C_DIS
LIN {X -0.087,Y -574.434,Z 1250.958,A 0.000,B 0.000,C 90.000,E1 28.437} C_DIS
LIN {X 0.212,Y -570.100,Z 1250.953,A 0.000,B 0.000,C 90.000,E1 27.590} C_DIS
LIN {X -0.126,Y -566.989,Z 1250.950,A 0.000,B 0.000,C 90.000,E1 27.078} C_DIS
LIN {X 0.275,Y -563.661,Z 1250.947,A 0.000,B 0.000,C 90.000,E1 26.488} C_DIS
LIN {X -0.204,Y -559.168,Z 1250.943,A 0.000,B 0.000,C 90.000,E1 25.848} C_DIS
LIN {X -0.006,Y -556.305,Z 1250.941,A 0.000,B 0.000,C 90.000,E1 25.412} C_DIS
LIN {X -0.322,Y -553.292,Z 1250.939,A 0.000,B 0.000,C 90.000,E1 25.027} C_DIS
LIN {X -0.045,Y -545.682,Z 1250.933,A 0.000,B 0.000,C 90.000,E1 24.027} C_DIS
LIN {X -0.173,Y -539.722,Z 1250.930,A 0.000,B 0.000,C 90.000,E1 23.334} C_DIS
LIN {X 0.019,Y -534.919,Z 1250.927,A 0.000,B 0.000,C 90.000,E1 22.770} C_DIS
LIN {X 0.207,Y -525.836,Z 1250.921,A 0.000,B 0.000,C 90.000,E1 21.770} C_DIS
LIN {X -0.076,Y -516.610,Z 1250.916,A 0.000,B 0.000,C 90.000,E1 20.844} C_DIS
LIN {X -0.007,Y -505.894,Z 1250.910,A 0.000,B 0.000,C 90.000,E1 19.758} C_DIS
LIN {X 0.190,Y -495.853,Z 1250.905,A 0.000,B 0.000,C 90.000,E1 18.779} C_DIS
LIN {X -0.019,Y -487.161,Z 1250.900,A 0.000,B 0.000,C 90.000,E1 18.000} C_DIS
LIN {X 0.028,Y -480.008,Z 1250.896,A 0.000,B 0.000,C 90.000,E1 17.347} C_DIS
LIN {X -0.018,Y -471.087,Z 1250.892,A 0.000,B 0.000,C 90.000,E1 16.567} C_DIS
LIN {X 0.216,Y -459.286,Z 1250.886,A 0.000,B 0.000,C 90.000,E1 15.481} C_DIS
LIN {X -0.086,Y -437.220,Z 1250.875,A 0.000,B 0.000,C 90.000,E1 13.467} C_DIS
LIN {X 0.130,Y -417.054,Z 1250.863,A 0.000,B 0.000,C 90.000,E1 11.366} C_DIS
LIN {X -0.125,Y -405.588,Z 1250.856,A 0.000,B 0.000,C 90.000,E1 10.141} C_DIS
LIN {X -0.155,Y -401.308,Z 1250.854,A 0.000,B 0.000,C 90.000,E1 9.670} C_DIS
LIN {X -0.159,Y -397.023,Z 1250.850,A 0.000,B 0.000,C 90.000,E1 9.095} C_DIS
LIN {X -0.134,Y -394.507,Z 1250.848,A 0.000,B 0.000,C 90.000,E1 8.624} C_DIS
LIN {X -0.172,Y -394.485,Z 1250.848,A 0.000,B 0.000,C 90.000,E1 8.624} C_DIS
LIN {X 0.191,Y -394.399,Z 1250.848,A 0.000,B 0.000,C 90.000,E1 8.511} C_DIS
LIN {X 0.153,Y -394.403,Z 1250.847,A 0.000,B 0.000,C 90.000,E1 8.511} C_DIS
LIN {X -0.022,Y -396.303,Z 1250.845,A 0.000,B 0.000,C 90.000,E1 8.106} C_DIS
LIN {X 0.023,Y -399.519,Z 1250.843,A 0.000,B 0.000,C 90.000,E1 7.757} C_DIS
LIN {X 0.150,Y -401.201,Z 1250.842,A 0.000,B 0.000,C 90.000,E1 7.587} C_DIS
LIN {X -0.093,Y -410.073,Z 1250.839,A 0.000,B 0.000,C 90.000,E1 7.004} C_DIS
LIN {X -0.002,Y -419.754,Z 1250.835,A 0.000,B 0.000,C 90.000,E1 6.315} C_DIS
LIN {X -0.126,Y -429.417,Z 1250.831,A 0.000,B 0.000,C 90.000,E1 5.625} C_DIS
LIN {X 0.002,Y -438.653,Z 1250.827,A 0.000,B 0.000,C 90.000,E1 4.878} C_DIS
LIN {X -0.110,Y -452.535,Z 1250.821,A 0.000,B 0.000,C 90.000,E1 3.784} C_DIS
LIN {X -0.160,Y -461.580,Z 1250.817,A 0.000,B 0.000,C 90.000,E1 3.037} C_DIS
LIN {X -0.166,Y -467.549,Z 1250.814,A 0.000,B 0.000,C 90.000,E1 2.522} C_DIS
LIN {X -0.243,Y -473.311,Z 1250.811,A 0.000,B 0.000,C 90.000,E1 2.007} C_DIS
LIN {X 0.196,Y -478.682,Z 1250.808,A 0.000,B 0.000,C 90.000,E1 1.432} C_DIS
LIN {X 0.032,Y -485.366,Z 1250.804,A 0.000,B 0.000,C 90.000,E1 0.745} C_DIS
LIN {X 0.000,Y -491.800,Z 1250.800,A 0.000,B 0.000,C 90.000,E1 360.000} C_DIS
LIN {X 0.035,Y -496.035,Z 1250.797,A 0.000,B 0.000,C 90.000,E1 359.484} C_DIS
LIN {X 0.132,Y -502.717,Z 1250.792,A 0.000,B 0.000,C 90.000,E1 358.568} C_DIS
LIN {X -0.083,Y -506.888,Z 1250.789,A 0.000,B 0.000,C 90.000,E1 357.993} C_DIS
LIN {X -0.077,Y -511.741,Z 1250.785,A 0.000,B 0.000,C 90.000,E1 357.249} C_DIS
LIN {X -0.005,Y -516.323,Z 1250.781,A 0.000,B 0.000,C 90.000,E1 356.502} C_DIS
LIN {X -0.112,Y -519.769,Z 1250.777,A 0.000,B 0.000,C 90.000,E1 355.927} C_DIS
LIN {X 0.042,Y -523.692,Z 1250.773,A 0.000,B 0.000,C 90.000,E1 355.179} C_DIS
LIN {X 0.231,Y -527.317,Z 1250.769,A 0.000,B 0.000,C 90.000,E1 354.432} C_DIS
LIN {X 0.208,Y -530.036,Z 1250.766,A 0.000,B 0.000,C 90.000,E1 353.856} C_DIS
LIN {X 0.203,Y -532.581,Z 1250.763,A 0.000,B 0.000,C 90.000,E1 353.280} C_DIS
LIN {X 0.257,Y -535.987,Z 1250.758,A 0.000,B 0.000,C 90.000,E1 352.413} C_DIS
LIN {X -0.187,Y -539.097,Z 1250.753,A 0.000,B 0.000,C 90.000,E1 351.602} C_DIS
LIN {X -0.068,Y -542.025,Z 1250.749,A 0.000,B 0.000,C 90.000,E1 350.735} C_DIS
LIN {X 0.173,Y -544.564,Z 1250.744,A 0.000,B 0.000,C 90.000,E1 349.859} C_DIS
LIN {X -0.097,Y -547.736,Z 1250.738,A 0.000,B 0.000,C 90.000,E1 348.757} C_DIS
LIN {X -0.224,Y -550.511,Z 1250.731,A 0.000,B 0.000,C 90.000,E1 347.645} C_DIS
LIN {X -0.068,Y -553.621,Z 1250.724,A 0.000,B 0.000,C 90.000,E1 346.228} C_DIS
LIN {X -0.244,Y -555.270,Z 1250.719,A 0.000,B 0.000,C 90.000,E1 345.408} C_DIS
LIN {X 0.141,Y -557.662,Z 1250.711,A 0.000,B 0.000,C 90.000,E1 343.976} C_DIS
LIN {X -0.256,Y -559.263,Z 1250.705,A 0.000,B 0.000,C 90.000,E1 342.906} C_DIS
LIN {X -0.065,Y -560.305,Z 1250.700,A 0.000,B 0.000,C 90.000,E1 342.054} C_DIS
LIN {X 0.272,Y -561.346,Z 1250.694,A 0.000,B 0.000,C 90.000,E1 340.913} C_DIS
LIN {X -0.036,Y -561.858,Z 1250.690,A 0.000,B 0.000,C 90.000,E1 340.115} C_DIS
LIN {X 0.191,Y -562.096,Z 1250.685,A 0.000,B 0.000,C 90.000,E1 339.263} C_DIS
LIN {X 0.099,Y -562.146,Z 1250.682,A 0.000,B 0.000,C 90.000,E1 338.720} C_DIS
LIN {X -0.204,Y -561.843,Z 1250.677,A 0.000,B 0.000,C 90.000,E1 337.922} C_DIS
LIN {X 0.223,Y -561.197,Z 1250.673,A 0.000,B 0.000,C 90.000,E1 337.050} C_DIS
LIN {X 0.130,Y -560.290,Z 1250.668,A 0.000,B 0.000,C 90.000,E1 336.230} C_DIS
LIN {X 0.235,Y -559.483,Z 1250.665,A 0.000,B 0.000,C 90.000,E1 335.665} C_DIS
LIN {X 0.128,Y -558.030,Z 1250.660,A 0.000,B 0.000,C 90.000,E1 334.845} C_DIS
LIN {X -0.207,Y -555.656,Z 1250.654,A 0.000,B 0.000,C 90.000,E1 333.768} C_DIS
LIN {X -0.141,Y -554.373,Z 1250.651,A 0.000,B 0.000,C 90.000,E1 333.204} C_DIS
LIN {X 0.164,Y -552.561,Z 1250.648,A 0.000,B 0.000,C 90.000,E1 332.615} C_DIS
LIN {X -0.059,Y -551.791,Z 1250.646,A 0.000,B 0.000,C 90.000,E1 332.359} C_DIS
LIN {X -0.003,Y -548.733,Z 1250.642,A 0.000,B 0.000,C 90.000,E1 331.513} C_DIS
LIN {X 0.265,Y -546.432,Z 1250.639,A 0.000,B 0.000,C 90.000,E1 330.923} C_DIS
LIN {X -0.088,Y -543.086,Z 1250.635,A 0.000,B 0.000,C 90.000,E1 330.255} C_DIS
LIN {X 0.000,Y -539.327,Z 1250.631,A 0.000,B 0.000,C 90.000,E1 329.537} C_DIS
LIN {X 0.046,Y -534.918,Z 1250.627,A 0.000,B 0.000,C 90.000,E1 328.820} C_DIS
LIN {X 0.304,Y -528.358,Z 1250.621,A 0.000,B 0.000,C 90.000,E1 327.788} C_DIS
LIN {X -0.243,Y -521.327,Z 1250.616,A 0.000,B 0.000,C 90.000,E1 326.834} C_DIS
LIN {X -0.086,Y -516.440,Z 1250.612,A 0.000,B 0.000,C 90.000,E1 326.087} C_DIS
LIN {X 0.146,Y -513.119,Z 1250.609,A 0.000,B 0.000,C 90.000,E1 325.515} C_DIS
LIN {X -0.301,Y -509.922,Z 1250.605,A 0.000,B 0.000,C 90.000,E1 324.975} C_DIS
LIN {X -0.017,Y -507.618,Z 1250.602,A 0.000,B 0.000,C 90.000,E1 324.356} C_DIS
LIN {X -0.177,Y -505.961,Z 1250.599,A 0.000,B 0.000,C 90.000,E1 323.783} C_DIS
LIN {X 0.250,Y -504.354,Z 1250.594,A 0.000,B 0.000,C 90.000,E1 322.844} C_DIS
LIN {X -0.074,Y -503.629,Z 1250.589,A 0.000,B 0.000,C 90.000,E1 321.984} C_DIS
LIN {X -0.147,Y -504.191,Z 1250.569,A 0.000,B 0.000,C 90.000,E1 318.405} C_DIS
LIN {X 0.001,Y -504.801,Z 1250.557,A 0.000,B 0.000,C 90.000,E1 316.296} C_DIS
LIN {X 0.189,Y -505.078,Z 1250.551,A 0.000,B 0.000,C 90.000,E1 315.081} C_DIS
LIN {X 0.119,Y -505.506,Z 1250.541,A 0.000,B 0.000,C 90.000,E1 313.299} C_DIS
LIN {X -0.037,Y -506.102,Z 1250.529,A 0.000,B 0.000,C 90.000,E1 311.229} C_DIS
LIN {X -0.014,Y -506.510,Z 1250.519,A 0.000,B 0.000,C 90.000,E1 309.439} C_DIS
LIN {X -0.087,Y -507.006,Z 1250.508,A 0.000,B 0.000,C 90.000,E1 307.363} C_DIS
LIN {X -0.075,Y -507.339,Z 1250.501,A 0.000,B 0.000,C 90.000,E1 306.171} C_DIS
LIN {X -0.050,Y -507.523,Z 1250.494,A 0.000,B 0.000,C 90.000,E1 304.978} C_DIS
LIN {X 0.198,Y -507.697,Z 1250.484,A 0.000,B 0.000,C 90.000,E1 303.166} C_DIS
LIN {X 0.159,Y -507.760,Z 1250.474,A 0.000,B 0.000,C 90.000,E1 301.386} C_DIS
LIN {X -0.089,Y -507.701,Z 1250.463,A 0.000,B 0.000,C 90.000,E1 299.333} C_DIS
LIN {X -0.176,Y -507.610,Z 1250.456,A 0.000,B 0.000,C 90.000,E1 298.153} C_DIS
LIN {X 0.268,Y -507.454,Z 1250.448,A 0.000,B 0.000,C 90.000,E1 296.616} C_DIS
LIN {X -0.236,Y -507.436,Z 1250.437,A 0.000,B 0.000,C 90.000,E1 294.591} C_DIS
LIN {X -0.203,Y -507.457,Z 1250.432,A 0.000,B 0.000,C 90.000,E1 293.695} C_DIS
LIN {X -0.087,Y -507.121,Z 1250.422,A 0.000,B 0.000,C 90.000,E1 291.897} C_DIS
LIN {X -0.167,Y -506.339,Z 1250.412,A 0.000,B 0.000,C 90.000,E1 290.120} C_DIS
LIN {X 0.147,Y -505.190,Z 1250.397,A 0.000,B 0.000,C 90.000,E1 287.402} C_DIS
LIN {X 0.239,Y -504.876,Z 1250.392,A 0.000,B 0.000,C 90.000,E1 286.496} C_DIS
LIN {X 0.190,Y -504.192,Z 1250.384,A 0.000,B 0.000,C 90.000,E1 285.009} C_DIS
LIN {X 0.002,Y -503.274,Z 1250.375,A 0.000,B 0.000,C 90.000,E1 283.536} C_DIS
LIN {X -0.202,Y -502.232,Z 1250.367,A 0.000,B 0.000,C 90.000,E1 282.063} C_DIS
LIN {X -0.041,Y -501.115,Z 1250.359,A 0.000,B 0.000,C 90.000,E1 280.546} C_DIS
LIN {X -0.057,Y -499.901,Z 1250.349,A 0.000,B 0.000,C 90.000,E1 278.746} C_DIS
LIN {X -0.252,Y -498.588,Z 1250.337,A 0.000,B 0.000,C 90.000,E1 276.663} C_DIS
LIN {X -0.050,Y -497.594,Z 1250.325,A 0.000,B 0.000,C 90.000,E1 274.531} C_DIS
LIN {X -0.069,Y -496.902,Z 1250.318,A 0.000,B 0.000,C 90.000,E1 273.326} C_DIS
LIN {X -0.214,Y -495.826,Z 1250.310,A 0.000,B 0.000,C 90.000,E1 271.833} C_DIS
LIN {X 0.004,Y -493.745,Z 1250.295,A 0.000,B 0.000,C 90.000,E1 269.083} C_DIS
LIN {X -0.222,Y -492.645,Z 1250.286,A 0.000,B 0.000,C 90.000,E1 267.593} C_DIS
LIN {X -0.158,Y -492.154,Z 1250.281,A 0.000,B 0.000,C 90.000,E1 266.674} C_DIS
LIN {X -0.049,Y -491.174,Z 1250.271,A 0.000,B 0.000,C 90.000,E1 264.837} C_DIS
LIN {X 0.040,Y -490.623,Z 1250.266,A 0.000,B 0.000,C 90.000,E1 263.913} C_DIS
LIN {X -0.161,Y -489.530,Z 1250.258,A 0.000,B 0.000,C 90.000,E1 262.413} C_DIS
LIN {X 0.162,Y -488.107,Z 1250.249,A 0.000,B 0.000,C 90.000,E1 260.849} C_DIS
LIN {X -0.063,Y -485.433,Z 1250.232,A 0.000,B 0.000,C 90.000,E1 257.813} C_DIS
LIN {X 0.230,Y -484.243,Z 1250.222,A 0.000,B 0.000,C 90.000,E1 255.936} C_DIS
LIN {X 0.124,Y -482.981,Z 1250.210,A 0.000,B 0.000,C 90.000,E1 253.795} C_DIS
LIN {X 0.122,Y -481.741,Z 1250.198,A 0.000,B 0.000,C 90.000,E1 251.638} C_DIS
LIN {X -0.056,Y -480.803,Z 1250.188,A 0.000,B 0.000,C 90.000,E1 249.806} C_DIS
LIN {X -0.247,Y -479.997,Z 1250.179,A 0.000,B 0.000,C 90.000,E1 248.284} C_DIS
LIN {X -0.109,Y -478.939,Z 1250.169,A 0.000,B 0.000,C 90.000,E1 246.410} C_DIS
LIN {X 0.021,Y -477.849,Z 1250.160,A 0.000,B 0.000,C 90.000,E1 244.845} C_DIS
LIN {X -0.099,Y -476.774,Z 1250.152,A 0.000,B 0.000,C 90.000,E1 243.307} C_DIS
LIN {X 0.216,Y -475.948,Z 1250.145,A 0.000,B 0.000,C 90.000,E1 242.025} C_DIS
LIN {X 0.276,Y -474.782,Z 1250.136,A 0.000,B 0.000,C 90.000,E1 240.461} C_DIS
LIN {X -0.106,Y -473.459,Z 1250.127,A 0.000,B 0.000,C 90.000,E1 238.948} C_DIS
LIN {X -0.070,Y -471.476,Z 1250.115,A 0.000,B 0.000,C 90.000,E1 236.755} C_DIS
LIN {X -0.244,Y -469.970,Z 1250.105,A 0.000,B 0.000,C 90.000,E1 234.895} C_DIS
LIN {X 0.060,Y -468.074,Z 1250.089,A 0.000,B 0.000,C 90.000,E1 232.029} C_DIS
LIN {X 0.207,Y -467.141,Z 1250.080,A 0.000,B 0.000,C 90.000,E1 230.436} C_DIS
LIN {X 0.269,Y -466.263,Z 1250.072,A 0.000,B 0.000,C 90.000,E1 228.852} C_DIS
LIN {X -0.035,Y -465.217,Z 1250.063,A 0.000,B 0.000,C 90.000,E1 227.310} C_DIS
LIN {X -0.104,Y -464.402,Z 1250.056,A 0.000,B 0.000,C 90.000,E1 226.053} C_DIS
LIN {X 0.160,Y -462.959,Z 1250.038,A 0.000,B 0.000,C 90.000,E1 222.852} C_DIS
LIN {X -0.071,Y -464.063,Z 1250.001,A 0.000,B 0.000,C 90.000,E1 216.217} C_DIS
LIN {X 0.094,Y -467.002,Z 1249.978,A 0.000,B 0.000,C 90.000,E1 212.084} C_DIS
LIN {X -0.016,Y -468.938,Z 1249.968,A 0.000,B 0.000,C 90.000,E1 210.207} C_DIS
LIN {X -0.214,Y -471.979,Z 1249.954,A 0.000,B 0.000,C 90.000,E1 207.719} C_DIS
LIN {X 0.163,Y -474.230,Z 1249.943,A 0.000,B 0.000,C 90.000,E1 205.796} C_DIS
LIN {X -0.069,Y -477.225,Z 1249.931,A 0.000,B 0.000,C 90.000,E1 203.643} C_DIS
LIN {X 0.024,Y -480.156,Z 1249.921,A 0.000,B 0.000,C 90.000,E1 201.770} C_DIS
LIN {X 0.153,Y -486.340,Z 1249.902,A 0.000,B 0.000,C 90.000,E1 198.362} C_DIS
LIN {X 0.050,Y -488.906,Z 1249.895,A 0.000,B 0.000,C 90.000,E1 197.149} C_DIS
LIN {X 0.193,Y -492.246,Z 1249.887,A 0.000,B 0.000,C 90.000,E1 195.607} C_DIS
LIN {X -0.168,Y -496.293,Z 1249.877,A 0.000,B 0.000,C 90.000,E1 193.828} C_DIS
LIN {X -0.224,Y -501.826,Z 1249.863,A 0.000,B 0.000,C 90.000,E1 191.422} C_DIS
LIN {X -0.166,Y -506.917,Z 1249.852,A 0.000,B 0.000,C 90.000,E1 189.321} C_DIS
LIN {X -0.099,Y -511.364,Z 1249.842,A 0.000,B 0.000,C 90.000,E1 187.530} C_DIS
LIN {X 0.104,Y -515.046,Z 1249.834,A 0.000,B 0.000,C 90.000,E1 186.030} C_DIS
LIN {X -0.115,Y -517.942,Z 1249.827,A 0.000,B 0.000,C 90.000,E1 184.878} C_DIS
LIN {X 0.137,Y -522.276,Z 1249.817,A 0.000,B 0.000,C 90.000,E1 183.094} C_DIS
LIN {X -0.104,Y -526.489,Z 1249.808,A 0.000,B 0.000,C 90.000,E1 181.375} C_DIS
LIN {X -0.221,Y -529.225,Z 1249.801,A 0.000,B 0.000,C 90.000,E1 180.229} C_DIS
LIN {X 0.223,Y -532.639,Z 1249.793,A 0.000,B 0.000,C 90.000,E1 178.740} C_DIS
LIN {X 0.214,Y -534.618,Z 1249.788,A 0.000,B 0.000,C 90.000,E1 177.879} C_DIS
LIN {X 0.240,Y -537.683,Z 1249.780,A 0.000,B 0.000,C 90.000,E1 176.445} C_DIS
LIN {X -0.239,Y -540.041,Z 1249.774,A 0.000,B 0.000,C 90.000,E1 175.355} C_DIS
LIN {X -0.037,Y -542.772,Z 1249.766,A 0.000,B 0.000,C 90.000,E1 173.913} C_DIS
LIN {X 0.237,Y -545.874,Z 1249.757,A 0.000,B 0.000,C 90.000,E1 172.186} C_DIS
LIN {X 0.083,Y -548.227,Z 1249.749,A 0.000,B 0.000,C 90.000,E1 170.792} C_DIS
LIN {X -0.137,Y -549.957,Z 1249.743,A 0.000,B 0.000,C 90.000,E1 169.690} C_DIS
LIN {X -0.118,Y -552.061,Z 1249.735,A 0.000,B 0.000,C 90.000,E1 168.285} C_DIS
LIN {X -0.060,Y -554.055,Z 1249.727,A 0.000,B 0.000,C 90.000,E1 166.881} C_DIS
LIN {X -0.254,Y -556.381,Z 1249.718,A 0.000,B 0.000,C 90.000,E1 165.227} C_DIS
LIN {X 0.171,Y -559.899,Z 1249.705,A 0.000,B 0.000,C 90.000,E1 162.960} C_DIS
LIN {X -0.027,Y -562.193,Z 1249.699,A 0.000,B 0.000,C 90.000,E1 161.873} C_DIS
LIN {X -0.055,Y -565.781,Z 1249.692,A 0.000,B 0.000,C 90.000,E1 160.496} C_DIS
LIN {X 0.016,Y -569.395,Z 1249.686,A 0.000,B 0.000,C 90.000,E1 159.390} C_DIS
LIN {X -0.025,Y -574.801,Z 1249.678,A 0.000,B 0.000,C 90.000,E1 158.028} C_DIS
LIN {X 0.001,Y -584.312,Z 1249.667,A 0.000,B 0.000,C 90.000,E1 155.997} C_DIS
LIN {X -0.012,Y -590.484,Z 1249.660,A 0.000,B 0.000,C 90.000,E1 154.793} C_DIS
LIN {X 0.075,Y -596.709,Z 1249.653,A 0.000,B 0.000,C 90.000,E1 153.589} C_DIS
LIN {X 0.138,Y -600.089,Z 1249.650,A 0.000,B 0.000,C 90.000,E1 152.922} C_DIS
LIN {X -0.023,Y -605.981,Z 1249.643,A 0.000,B 0.000,C 90.000,E1 151.769} C_DIS
LIN {X -0.159,Y -609.143,Z 1249.640,A 0.000,B 0.000,C 90.000,E1 151.129} C_DIS
LIN {X 0.095,Y -614.615,Z 1249.633,A 0.000,B 0.000,C 90.000,E1 149.950} C_DIS
LIN {X 0.074,Y -620.055,Z 1249.627,A 0.000,B 0.000,C 90.000,E1 148.791} C_DIS
LIN {X -0.182,Y -624.817,Z 1249.621,A 0.000,B 0.000,C 90.000,E1 147.788} C_DIS
LIN {X 0.141,Y -628.156,Z 1249.617,A 0.000,B 0.000,C 90.000,E1 146.993} C_DIS
LIN {X -0.205,Y -632.425,Z 1249.611,A 0.000,B 0.000,C 90.000,E1 146.008} C_DIS
LIN {X 0.020,Y -635.428,Z 1249.607,A 0.000,B 0.000,C 90.000,E1 145.229} C_DIS
LIN {X -0.198,Y -640.129,Z 1249.600,A 0.000,B 0.000,C 90.000,E1 143.989} C_DIS
LIN {X 0.000,Y -643.457,Z 1249.594,A 0.000,B 0.000,C 90.000,E1 142.970} C_DIS
LIN {X 0.342,Y -645.796,Z 1249.590,A 0.000,B 0.000,C 90.000,E1 142.190} C_DIS
LIN {X 0.141,Y -649.384,Z 1249.583,A 0.000,B 0.000,C 90.000,E1 140.964} C_DIS
LIN {X -0.039,Y -652.090,Z 1249.578,A 0.000,B 0.000,C 90.000,E1 139.989} C_DIS
LIN {X 0.219,Y -655.973,Z 1249.570,A 0.000,B 0.000,C 90.000,E1 138.485} C_DIS
LIN {X -0.400,Y -659.075,Z 1249.563,A 0.000,B 0.000,C 90.000,E1 137.310} C_DIS
LIN {X -0.076,Y -663.907,Z 1249.552,A 0.000,B 0.000,C 90.000,E1 135.324} C_DIS
LIN {X -0.103,Y -668.480,Z 1249.542,A 0.000,B 0.000,C 90.000,E1 133.623} C_DIS
LIN {X -0.017,Y -672.437,Z 1249.534,A 0.000,B 0.000,C 90.000,E1 132.162} C_DIS
LIN {X 0.131,Y -675.680,Z 1249.528,A 0.000,B 0.000,C 90.000,E1 130.943} C_DIS
LIN {X 0.331,Y -678.868,Z 1249.521,A 0.000,B 0.000,C 90.000,E1 129.725} C_DIS
LIN {X -0.220,Y -683.230,Z 1249.512,A 0.000,B 0.000,C 90.000,E1 128.096} C_DIS
LIN {X -0.182,Y -686.932,Z 1249.504,A 0.000,B 0.000,C 90.000,E1 126.664} C_DIS
LIN {X -0.304,Y -689.205,Z 1249.498,A 0.000,B 0.000,C 90.000,E1 125.724} C_DIS
LIN {X -0.204,Y -691.899,Z 1249.492,A 0.000,B 0.000,C 90.000,E1 124.532} C_DIS
LIN {X -0.095,Y -693.929,Z 1249.487,A 0.000,B 0.000,C 90.000,E1 123.579} C_DIS
LIN {X 0.312,Y -696.826,Z 1249.479,A 0.000,B 0.000,C 90.000,E1 122.133} C_DIS
LIN {X -0.223,Y -699.022,Z 1249.472,A 0.000,B 0.000,C 90.000,E1 121.003} C_DIS
LIN {X 0.237,Y -701.116,Z 1249.466,A 0.000,B 0.000,C 90.000,E1 119.795} C_DIS
LIN {X 0.100,Y -702.544,Z 1249.460,A 0.000,B 0.000,C 90.000,E1 118.871} C_DIS
LIN {X -0.354,Y -703.753,Z 1249.455,A 0.000,B 0.000,C 90.000,E1 117.975} C_DIS
LIN {X 0.162,Y -704.662,Z 1249.450,A 0.000,B 0.000,C 90.000,E1 117.001} C_DIS
LIN {X 0.082,Y -705.103,Z 1249.446,A 0.000,B 0.000,C 90.000,E1 116.309} C_DIS
LIN {X 0.317,Y -705.220,Z 1249.442,A 0.000,B 0.000,C 90.000,E1 115.591} C_DIS
LIN {X -0.044,Y -705.105,Z 1249.440,A 0.000,B 0.000,C 90.000,E1 115.155} C_DIS
LIN {X -0.108,Y -704.742,Z 1249.437,A 0.000,B 0.000,C 90.000,E1 114.695} C_DIS
LIN {X 0.171,Y -704.033,Z 1249.435,A 0.000,B 0.000,C 90.000,E1 114.207} C_DIS
LIN {X -0.188,Y -703.609,Z 1249.433,A 0.000,B 0.000,C 90.000,E1 114.003} C_DIS
LIN {X 0.089,Y -701.656,Z 1249.431,A 0.000,B 0.000,C 90.000,E1 113.515} C_DIS
LIN {X 0.363,Y -700.446,Z 1249.429,A 0.000,B 0.000,C 90.000,E1 113.259} C_DIS
LIN {X -0.022,Y -696.157,Z 1249.427,A 0.000,B 0.000,C 90.000,E1 112.823} C_DIS
LIN {X 0.105,Y -694.882,Z 1249.426,A 0.000,B 0.000,C 90.000,E1 112.695} C_DIS
LIN {X -0.036,Y -692.851,Z 1249.426,A 0.000,B 0.000,C 90.000,E1 112.589} C_DIS
LIN {X 0.037,Y -687.935,Z 1249.425,A 0.000,B 0.000,C 90.000,E1 112.408} C_DIS
LIN {X 0.226,Y -686.012,Z 1249.424,A 0.000,B 0.000,C 90.000,E1 112.333} C_DIS
LIN {X -0.157,Y -677.229,Z 1249.424,A 0.000,B 0.000,C 90.000,E1 112.259} C_DIS
LIN {X -0.183,Y -626.353,Z 1249.424,A 0.000,B 0.000,C 90.000,E1 112.259} C_DIS
LIN {X 0.030,Y -625.541,Z 1249.423,A 0.000,B 0.000,C 90.000,E1 112.206} C_DIS
LIN {X -0.299,Y -622.551,Z 1249.422,A 0.000,B 0.000,C 90.000,E1 112.025} C_DIS
LIN {X -0.335,Y -622.523,Z 1249.422,A 0.000,B 0.000,C 90.000,E1 112.025} C_DIS
LIN {X 0.229,Y -622.140,Z 1249.422,A 0.000,B 0.000,C 90.000,E1 111.897} C_DIS
LIN {X 0.193,Y -622.131,Z 1249.422,A 0.000,B 0.000,C 90.000,E1 111.897} C_DIS
LIN {X 0.154,Y -622.835,Z 1249.420,A 0.000,B 0.000,C 90.000,E1 111.589} C_DIS
LIN {X 0.051,Y -623.937,Z 1249.419,A 0.000,B 0.000,C 90.000,E1 111.354} C_DIS
LIN {X -0.020,Y -628.739,Z 1249.414,A 0.000,B 0.000,C 90.000,E1 110.482} C_DIS
LIN {X -0.228,Y -631.656,Z 1249.411,A 0.000,B 0.000,C 90.000,E1 109.993} C_DIS
LIN {X 0.188,Y -634.882,Z 1249.407,A 0.000,B 0.000,C 90.000,E1 109.322} C_DIS
LIN {X 0.291,Y -640.801,Z 1249.401,A 0.000,B 0.000,C 90.000,E1 108.055} C_DIS
LIN {X -0.316,Y -646.741,Z 1249.394,A 0.000,B 0.000,C 90.000,E1 106.858} C_DIS
LIN {X 0.060,Y -650.158,Z 1249.389,A 0.000,B 0.000,C 90.000,E1 106.079} C_DIS
LIN {X -0.334,Y -653.174,Z 1249.385,A 0.000,B 0.000,C 90.000,E1 105.371} C_DIS
LIN {X 0.222,Y -654.902,Z 1249.383,A 0.000,B 0.000,C 90.000,E1 104.828} C_DIS
LIN {X -0.127,Y -657.060,Z 1249.378,A 0.000,B 0.000,C 90.000,E1 104.120} C_DIS
LIN {X 0.291,Y -658.152,Z 1249.376,A 0.000,B 0.000,C 90.000,E1 103.592} C_DIS
LIN {X 0.078,Y -659.002,Z 1249.373,A 0.000,B 0.000,C 90.000,E1 103.119} C_DIS
LIN {X -0.234,Y -659.844,Z 1249.369,A 0.000,B 0.000,C 90.000,E1 102.411} C_DIS
LIN {X 0.205,Y -659.934,Z 1249.366,A 0.000,B 0.000,C 90.000,E1 101.883} C_DIS
LIN {X -0.133,Y -659.694,Z 1249.363,A 0.000,B 0.000,C 90.000,E1 101.422} C_DIS
LIN {X -0.236,Y -659.537,Z 1249.362,A 0.000,B 0.000,C 90.000,E1 101.186} C_DIS
LIN {X 0.202,Y -658.935,Z 1249.359,A 0.000,B 0.000,C 90.000,E1 100.658} C_DIS
LIN {X -0.132,Y -658.001,Z 1249.357,A 0.000,B 0.000,C 90.000,E1 100.197} C_DIS
LIN {X 0.291,Y -656.801,Z 1249.354,A 0.000,B 0.000,C 90.000,E1 99.670} C_DIS
LIN {X 0.067,Y -656.111,Z 1249.353,A 0.000,B 0.000,C 90.000,E1 99.443} C_DIS
LIN {X -0.172,Y -654.382,Z 1249.350,A 0.000,B 0.000,C 90.000,E1 98.973} C_DIS
LIN {X 0.120,Y -652.244,Z 1249.347,A 0.000,B 0.000,C 90.000,E1 98.454} C_DIS
LIN {X -0.269,Y -649.126,Z 1249.344,A 0.000,B 0.000,C 90.000,E1 97.871} C_DIS
LIN {X -0.133,Y -645.430,Z 1249.340,A 0.000,B 0.000,C 90.000,E1 97.239} C_DIS
LIN {X 0.099,Y -642.065,Z 1249.337,A 0.000,B 0.000,C 90.000,E1 96.720} C_DIS
LIN {X 0.308,Y -638.362,Z 1249.335,A 0.000,B 0.000,C 90.000,E1 96.201} C_DIS
LIN {X -0.234,Y -633.087,Z 1249.331,A 0.000,B 0.000,C 90.000,E1 95.625} C_DIS
LIN {X -0.035,Y -628.338,Z 1249.328,A 0.000,B 0.000,C 90.000,E1 95.106} C_DIS
LIN {X -0.137,Y -623.439,Z 1249.326,A 0.000,B 0.000,C 90.000,E1 94.645} C_DIS
LIN {X 0.305,Y -616.768,Z 1249.323,A 0.000,B 0.000,C 90.000,E1 94.012} C_DIS
LIN {X -0.287,Y -609.598,Z 1249.319,A 0.000,B 0.000,C 90.000,E1 93.498} C_DIS
LIN {X 0.271,Y -602.035,Z 1249.316,A 0.000,B 0.000,C 90.000,E1 92.922} C_DIS
LIN {X -0.130,Y -594.176,Z 1249.314,A 0.000,B 0.000,C 90.000,E1 92.465} C_DIS
LIN {X -0.127,Y -589.309,Z 1249.312,A 0.000,B 0.000,C 90.000,E1 92.178} C_DIS
LIN {X -0.167,Y -582.423,Z 1249.310,A 0.000,B 0.000,C 90.000,E1 91.835} C_DIS
LIN {X 0.157,Y -571.524,Z 1249.308,A 0.000,B 0.000,C 90.000,E1 91.375} C_DIS
LIN {X -0.005,Y -569.047,Z 1249.307,A 0.000,B 0.000,C 90.000,E1 91.260} C_DIS
LIN {X 0.012,Y -567.460,Z 1249.306,A 0.000,B 0.000,C 90.000,E1 91.146} C_DIS
LIN {X -0.026,Y -567.419,Z 1249.306,A 0.000,B 0.000,C 90.000,E1 91.146} C_DIS
LIN {X -0.214,Y -567.069,Z 1249.306,A 0.000,B 0.000,C 90.000,E1 91.088} C_DIS
LIN {X -0.208,Y -566.796,Z 1249.304,A 0.000,B 0.000,C 90.000,E1 90.745} C_DIS
LIN {X 0.015,Y -566.896,Z 1249.301,A 0.000,B 0.000,C 90.000,E1 90.115} C_DIS
LIN {X 0.165,Y -568.101,Z 1249.292,A 0.000,B 0.000,C 90.000,E1 88.453} C_DIS
LIN {X -0.068,Y -569.612,Z 1249.281,A 0.000,B 0.000,C 90.000,E1 86.560} C_DIS
LIN {X 0.035,Y -571.970,Z 1249.267,A 0.000,B 0.000,C 90.000,E1 84.090} C_DIS
LIN {X -0.115,Y -573.648,Z 1249.258,A 0.000,B 0.000,C 90.000,E1 82.470} C_DIS
LIN {X -0.221,Y -575.325,Z 1249.249,A 0.000,B 0.000,C 90.000,E1 80.849} C_DIS
LIN {X -0.056,Y -576.329,Z 1249.243,A 0.000,B 0.000,C 90.000,E1 79.746} C_DIS
LIN {X -0.028,Y -577.552,Z 1249.234,A 0.000,B 0.000,C 90.000,E1 78.117} C_DIS
LIN {X 0.268,Y -578.689,Z 1249.225,A 0.000,B 0.000,C 90.000,E1 76.464} C_DIS
LIN {X -0.330,Y -579.564,Z 1249.218,A 0.000,B 0.000,C 90.000,E1 75.172} C_DIS
LIN {X 0.161,Y -580.506,Z 1249.208,A 0.000,B 0.000,C 90.000,E1 73.504} C_DIS
LIN {X 0.109,Y -581.412,Z 1249.199,A 0.000,B 0.000,C 90.000,E1 71.891} C_DIS
LIN {X 0.047,Y -582.276,Z 1249.192,A 0.000,B 0.000,C 90.000,E1 70.550} C_DIS
LIN {X -0.219,Y -583.744,Z 1249.179,A 0.000,B 0.000,C 90.000,E1 68.156} C_DIS
LIN {X -0.348,Y -585.840,Z 1249.164,A 0.000,B 0.000,C 90.000,E1 65.485} C_DIS
LIN {X -0.123,Y -587.414,Z 1249.153,A 0.000,B 0.000,C 90.000,E1 63.589} C_DIS
LIN {X -0.127,Y -589.188,Z 1249.143,A 0.000,B 0.000,C 90.000,E1 61.719} C_DIS
LIN {X -0.212,Y -590.868,Z 1249.134,A 0.000,B 0.000,C 90.000,E1 60.127} C_DIS
LIN {X -0.054,Y -592.804,Z 1249.124,A 0.000,B 0.000,C 90.000,E1 58.250} C_DIS
LIN {X 0.037,Y -594.108,Z 1249.116,A 0.000,B 0.000,C 90.000,E1 56.914} C_DIS
LIN {X 0.196,Y -595.547,Z 1249.107,A 0.000,B 0.000,C 90.000,E1 55.308} C_DIS
LIN {X 0.157,Y -596.707,Z 1249.100,A 0.000,B 0.000,C 90.000,E1 53.989} C_DIS
LIN {X -0.121,Y -598.018,Z 1249.091,A 0.000,B 0.000,C 90.000,E1 52.431} C_DIS
LIN {X 0.119,Y -599.033,Z 1249.084,A 0.000,B 0.000,C 90.000,E1 51.090} C_DIS
LIN {X -0.236,Y -599.628,Z 1249.078,A 0.000,B 0.000,C 90.000,E1 50.070} C_DIS
LIN {X 0.033,Y -600.253,Z 1249.071,A 0.000,B 0.000,C 90.000,E1 48.728} C_DIS
LIN {X 0.260,Y -600.792,Z 1249.063,A 0.000,B 0.000,C 90.000,E1 47.391} C_DIS
LIN {X 0.294,Y -601.091,Z 1249.055,A 0.000,B 0.000,C 90.000,E1 45.810} C_DIS
LIN {X 0.319,Y -601.194,Z 1249.049,A 0.000,B 0.000,C 90.000,E1 44.757} C_DIS
LIN {X 0.341,Y -601.033,Z 1249.043,A 0.000,B 0.000,C 90.000,E1 43.704} C_DIS
LIN {X -0.055,Y -600.724,Z 1249.037,A 0.000,B 0.000,C 90.000,E1 42.690} C_DIS
LIN {X -0.006,Y -600.358,Z 1249.031,A 0.000,B 0.000,C 90.000,E1 41.634} C_DIS
LIN {X -0.411,Y -599.880,Z 1249.026,A 0.000,B 0.000,C 90.000,E1 40.620} C_DIS
LIN {X -0.151,Y -599.446,Z 1249.021,A 0.000,B 0.000,C 90.000,E1 39.806} C_DIS
LIN {X -0.122,Y -598.767,Z 1249.015,A 0.000,B 0.000,C 90.000,E1 38.749} C_DIS
LIN {X -0.008,Y -597.864,Z 1249.009,A 0.000,B 0.000,C 90.000,E1 37.684} C_DIS
LIN {X -0.143,Y -596.397,Z 1249.002,A 0.000,B 0.000,C 90.000,E1 36.377} C_DIS
LIN {X -0.058,Y -594.918,Z 1248.996,A 0.000,B 0.000,C 90.000,E1 35.311} C_DIS
LIN {X 0.000,Y -593.063,Z 1248.990,A 0.000,B 0.000,C 90.000,E1 34.246} C_DIS
LIN {X -0.020,Y -591.521,Z 1248.986,A 0.000,B 0.000,C 90.000,E1 33.452} C_DIS
LIN {X -0.222,Y -589.718,Z 1248.981,A 0.000,B 0.000,C 90.000,E1 32.673} C_DIS
LIN {X -0.265,Y -587.554,Z 1248.977,A 0.000,B 0.000,C 90.000,E1 31.878} C_DIS
LIN {X -0.022,Y -585.027,Z 1248.973,A 0.000,B 0.000,C 90.000,E1 31.052} C_DIS
LIN {X 0.020,Y -583.170,Z 1248.970,A 0.000,B 0.000,C 90.000,E1 30.512} C_DIS
LIN {X -0.089,Y -580.006,Z 1248.965,A 0.000,B 0.000,C 90.000,E1 29.716} C_DIS
LIN {X -0.007,Y -576.437,Z 1248.961,A 0.000,B 0.000,C 90.000,E1 28.899} C_DIS
LIN {X -0.188,Y -572.335,Z 1248.956,A 0.000,B 0.000,C 90.000,E1 28.103} C_DIS
LIN {X 0.258,Y -569.353,Z 1248.953,A 0.000,B 0.000,C 90.000,E1 27.513} C_DIS
LIN {X -0.088,Y -566.189,Z 1248.950,A 0.000,B 0.000,C 90.000,E1 27.001} C_DIS
LIN {X 0.054,Y -562.824,Z 1248.947,A 0.000,B 0.000,C 90.000,E1 26.437} C_DIS
LIN {X 0.317,Y -558.298,Z 1248.943,A 0.000,B 0.000,C 90.000,E1 25.720} C_DIS
LIN {X -0.207,Y -553.387,Z 1248.939,A 0.000,B 0.000,C 90.000,E1 25.079} C_DIS
LIN {X 0.110,Y -546.834,Z 1248.935,A 0.000,B 0.000,C 90.000,E1 24.207} C_DIS
LIN {X 0.241,Y -543.395,Z 1248.932,A 0.000,B 0.000,C 90.000,E1 23.770} C_DIS
LIN {X 0.222,Y -538.545,Z 1248.929,A 0.000,B 0.000,C 90.000,E1 23.206} C_DIS
LIN {X 0.201,Y -533.518,Z 1248.926,A 0.000,B 0.000,C 90.000,E1 22.642} C_DIS
LIN {X -0.205,Y -525.683,Z 1248.921,A 0.000,B 0.000,C 90.000,E1 21.844} C_DIS
LIN {X 0.010,Y -516.458,Z 1248.916,A 0.000,B 0.000,C 90.000,E1 20.865} C_DIS
LIN {X -0.185,Y -505.745,Z 1248.910,A 0.000,B 0.000,C 90.000,E1 19.812} C_DIS
LIN {X -0.105,Y -495.776,Z 1248.905,A 0.000,B 0.000,C 90.000,E1 18.852} C_DIS
LIN {X -0.165,Y -487.091,Z 1248.900,A 0.000,B 0.000,C 90.000,E1 18.055} C_DIS
LIN {X -0.196,Y -479.816,Z 1248.897,A 0.000,B 0.000,C 90.000,E1 17.402} C_DIS
LIN {X -0.024,Y -463.889,Z 1248.889,A 0.000,B 0.000,C 90.000,E1 15.969} C_DIS
LIN {X 0.163,Y -447.726,Z 1248.881,A 0.000,B 0.000,C 90.000,E1 14.481} C_DIS
LIN {X -0.203,Y -424.459,Z 1248.868,A 0.000,B 0.000,C 90.000,E1 12.243} C_DIS
LIN {X -0.062,Y -407.377,Z 1248.858,A 0.000,B 0.000,C 90.000,E1 10.366} C_DIS
LIN {X -0.070,Y -401.556,Z 1248.854,A 0.000,B 0.000,C 90.000,E1 9.726} C_DIS
LIN {X 0.067,Y -396.563,Z 1248.850,A 0.000,B 0.000,C 90.000,E1 9.029} C_DIS
LIN {X 0.115,Y -394.499,Z 1248.848,A 0.000,B 0.000,C 90.000,E1 8.624} C_DIS
LIN {X 0.077,Y -394.482,Z 1248.848,A 0.000,B 0.000,C 90.000,E1 8.624} C_DIS
LIN {X -0.178,Y -394.369,Z 1248.848,A 0.000,B 0.000,C 90.000,E1 8.568} C_DIS
LIN {X 0.174,Y -394.368,Z 1248.848,A 0.000,B 0.000,C 90.000,E1 8.511} C_DIS
LIN {X -0.117,Y -396.416,Z 1248.845,A 0.000,B 0.000,C 90.000,E1 8.106} C_DIS
LIN {X -0.063,Y -400.835,Z 1248.842,A 0.000,B 0.000,C 90.000,E1 7.644} C_DIS
LIN {X 0.077,Y -406.159,Z 1248.840,A 0.000,B 0.000,C 90.000,E1 7.239} C_DIS
LIN {X -0.071,Y -412.454,Z 1248.838,A 0.000,B 0.000,C 90.000,E1 6.834} C_DIS
LIN {X 0.024,Y -423.566,Z 1248.834,A 0.000,B 0.000,C 90.000,E1 6.030} C_DIS
LIN {X -0.117,Y -431.475,Z 1248.830,A 0.000,B 0.000,C 90.000,E1 5.454} C_DIS
LIN {X -0.094,Y -440.910,Z 1248.826,A 0.000,B 0.000,C 90.000,E1 4.702} C_DIS
LIN {X 0.032,Y -450.055,Z 1248.822,A 0.000,B 0.000,C 90.000,E1 3.955} C_DIS
LIN {X 0.090,Y -459.134,Z 1248.818,A 0.000,B 0.000,C 90.000,E1 3.212} C_DIS
LIN {X -0.064,Y -468.104,Z 1248.814,A 0.000,B 0.000,C 90.000,E1 2.465} C_DIS
LIN {X -0.015,Y -472.536,Z 1248.812,A 0.000,B 0.000,C 90.000,E1 2.064} C_DIS
LIN {X 0.141,Y -479.423,Z 1248.808,A 0.000,B 0.000,C 90.000,E1 1.375} C_DIS
LIN {X 0.134,Y -484.898,Z 1248.805,A 0.000,B 0.000,C 90.000,E1 0.802} C_DIS
LIN {X 0.205,Y -489.896,Z 1248.802,A 0.000,B 0.000,C 90.000,E1 0.229} C_DIS
LIN {X 0.104,Y -496.227,Z 1248.797,A 0.000,B 0.000,C 90.000,E1 359.484} C_DIS
LIN {X 0.204,Y -502.960,Z 1248.792,A 0.000,B 0.000,C 90.000,E1 358.568} C_DIS
LIN {X 0.053,Y -507.139,Z 1248.789,A 0.000,B 0.000,C 90.000,E1 357.993} C_DIS
LIN {X 0.062,Y -512.001,Z 1248.785,A 0.000,B 0.000,C 90.000,E1 357.249} C_DIS
LIN {X 0.138,Y -516.618,Z 1248.781,A 0.000,B 0.000,C 90.000,E1 356.502} C_DIS
LIN {X 0.034,Y -520.072,Z 1248.777,A 0.000,B 0.000,C 90.000,E1 355.927} C_DIS
LIN {X 0.192,Y -524.033,Z 1248.773,A 0.000,B 0.000,C 90.000,E1 355.179} C_DIS
LIN {X -0.139,Y -527.660,Z 1248.769,A 0.000,B 0.000,C 90.000,E1 354.489} C_DIS
LIN {X -0.162,Y -530.385,Z 1248.766,A 0.000,B 0.000,C 90.000,E1 353.913} C_DIS
LIN {X -0.165,Y -532.936,Z 1248.763,A 0.000,B 0.000,C 90.000,E1 353.337} C_DIS
LIN {X -0.154,Y -535.292,Z 1248.760,A 0.000,B 0.000,C 90.000,E1 352.761} C_DIS
LIN {X -0.075,Y -538.483,Z 1248.755,A 0.000,B 0.000,C 90.000,E1 351.894} C_DIS
LIN {X 0.109,Y -542.391,Z 1248.749,A 0.000,B 0.000,C 90.000,E1 350.735} C_DIS
LIN {X -0.183,Y -544.931,Z 1248.744,A 0.000,B 0.000,C 90.000,E1 349.916} C_DIS
LIN {X 0.091,Y -548.107,Z 1248.738,A 0.000,B 0.000,C 90.000,E1 348.757} C_DIS
LIN {X -0.138,Y -550.227,Z 1248.733,A 0.000,B 0.000,C 90.000,E1 347.937} C_DIS
LIN {X 0.193,Y -552.156,Z 1248.728,A 0.000,B 0.000,C 90.000,E1 347.061} C_DIS
LIN {X 0.255,Y -554.582,Z 1248.722,A 0.000,B 0.000,C 90.000,E1 345.936} C_DIS
LIN {X 0.230,Y -556.216,Z 1248.717,A 0.000,B 0.000,C 90.000,E1 345.102} C_DIS
LIN {X -0.050,Y -558.554,Z 1248.710,A 0.000,B 0.000,C 90.000,E1 343.740} C_DIS
LIN {X -0.034,Y -559.732,Z 1248.705,A 0.000,B 0.000,C 90.000,E1 342.906} C_DIS
LIN {X -0.240,Y -561.095,Z 1248.699,A 0.000,B 0.000,C 90.000,E1 341.819} C_DIS
LIN {X 0.105,Y -562.090,Z 1248.693,A 0.000,B 0.000,C 90.000,E1 340.678} C_DIS
LIN {X -0.199,Y -562.562,Z 1248.688,A 0.000,B 0.000,C 90.000,E1 339.880} C_DIS
LIN {X -0.174,Y -562.762,Z 1248.682,A 0.000,B 0.000,C 90.000,E1 338.773} C_DIS
LIN {X -0.265,Y -562.654,Z 1248.679,A 0.000,B 0.000,C 90.000,E1 338.230} C_DIS
LIN {X -0.147,Y -562.389,Z 1248.676,A 0.000,B 0.000,C 90.000,E1 337.667} C_DIS
LIN {X 0.288,Y -561.666,Z 1248.671,A 0.000,B 0.000,C 90.000,E1 336.794} C_DIS
LIN {X -0.024,Y -560.737,Z 1248.667,A 0.000,B 0.000,C 90.000,E1 335.997} C_DIS
LIN {X 0.080,Y -559.865,Z 1248.664,A 0.000,B 0.000,C 90.000,E1 335.433} C_DIS
LIN {X 0.210,Y -558.327,Z 1248.659,A 0.000,B 0.000,C 90.000,E1 334.588} C_DIS
LIN {X 0.161,Y -555.337,Z 1248.651,A 0.000,B 0.000,C 90.000,E1 333.204} C_DIS
LIN {X 0.252,Y -552.779,Z 1248.647,A 0.000,B 0.000,C 90.000,E1 332.359} C_DIS
LIN {X -0.166,Y -549.779,Z 1248.642,A 0.000,B 0.000,C 90.000,E1 331.563} C_DIS
LIN {X 0.113,Y -547.523,Z 1248.639,A 0.000,B 0.000,C 90.000,E1 330.973} C_DIS
LIN {X 0.120,Y -543.491,Z 1248.634,A 0.000,B 0.000,C 90.000,E1 330.127} C_DIS
LIN {X -0.123,Y -540.509,Z 1248.631,A 0.000,B 0.000,C 90.000,E1 329.587} C_DIS
LIN {X -0.200,Y -535.211,Z 1248.626,A 0.000,B 0.000,C 90.000,E1 328.742} C_DIS
LIN {X 0.065,Y -528.619,Z 1248.621,A 0.000,B 0.000,C 90.000,E1 327.709} C_DIS
LIN {X 0.128,Y -522.463,Z 1248.616,A 0.000,B 0.000,C 90.000,E1 326.834} C_DIS
LIN {X -0.138,Y -517.466,Z 1248.612,A 0.000,B 0.000,C 90.000,E1 326.135} C_DIS
LIN {X -0.020,Y -512.919,Z 1248.608,A 0.000,B 0.000,C 90.000,E1 325.388} C_DIS
LIN {X -0.281,Y -510.450,Z 1248.605,A 0.000,B 0.000,C 90.000,E1 324.975} C_DIS
LIN {X 0.050,Y -509.177,Z 1248.604,A 0.000,B 0.000,C 90.000,E1 324.642} C_DIS
LIN {X -0.040,Y -508.033,Z 1248.602,A 0.000,B 0.000,C 90.000,E1 324.356} C_DIS
LIN {X -0.223,Y -506.317,Z 1248.599,A 0.000,B 0.000,C 90.000,E1 323.783} C_DIS
LIN {X 0.208,Y -504.694,Z 1248.594,A 0.000,B 0.000,C 90.000,E1 322.844} C_DIS
LIN {X -0.112,Y -503.954,Z 1248.589,A 0.000,B 0.000,C 90.000,E1 321.984} C_DIS
LIN {X -0.129,Y -503.848,Z 1248.584,A 0.000,B 0.000,C 90.000,E1 321.090} C_DIS
LIN {X -0.172,Y -504.591,Z 1248.569,A 0.000,B 0.000,C 90.000,E1 318.405} C_DIS
LIN {X -0.012,Y -505.201,Z 1248.557,A 0.000,B 0.000,C 90.000,E1 316.296} C_DIS
LIN {X 0.182,Y -505.505,Z 1248.551,A 0.000,B 0.000,C 90.000,E1 315.081} C_DIS
LIN {X 0.122,Y -505.933,Z 1248.541,A 0.000,B 0.000,C 90.000,E1 313.299} C_DIS
LIN {X -0.140,Y -506.373,Z 1248.532,A 0.000,B 0.000,C 90.000,E1 311.838} C_DIS
LIN {X -0.009,Y -506.790,Z 1248.524,A 0.000,B 0.000,C 90.000,E1 310.334} C_DIS
LIN {X 0.232,Y -507.035,Z 1248.517,A 0.000,B 0.000,C 90.000,E1 309.116} C_DIS
LIN {X -0.051,Y -507.523,Z 1248.508,A 0.000,B 0.000,C 90.000,E1 307.363} C_DIS
LIN {X -0.030,Y -507.841,Z 1248.501,A 0.000,B 0.000,C 90.000,E1 306.171} C_DIS
LIN {X -0.093,Y -508.058,Z 1248.493,A 0.000,B 0.000,C 90.000,E1 304.692} C_DIS
LIN {X 0.263,Y -508.256,Z 1248.484,A 0.000,B 0.000,C 90.000,E1 303.166} C_DIS
LIN {X -0.091,Y -508.342,Z 1248.476,A 0.000,B 0.000,C 90.000,E1 301.720} C_DIS
LIN {X 0.118,Y -508.290,Z 1248.465,A 0.000,B 0.000,C 90.000,E1 299.617} C_DIS
LIN {X 0.047,Y -508.256,Z 1248.458,A 0.000,B 0.000,C 90.000,E1 298.437} C_DIS
LIN {X -0.074,Y -508.059,Z 1248.448,A 0.000,B 0.000,C 90.000,E1 296.668} C_DIS
LIN {X -0.107,Y -508.095,Z 1248.437,A 0.000,B 0.000,C 90.000,E1 294.591} C_DIS
LIN {X -0.067,Y -508.090,Z 1248.432,A 0.000,B 0.000,C 90.000,E1 293.695} C_DIS
LIN {X -0.038,Y -507.848,Z 1248.423,A 0.000,B 0.000,C 90.000,E1 292.206} C_DIS
LIN {X 0.261,Y -507.501,Z 1248.418,A 0.000,B 0.000,C 90.000,E1 291.280} C_DIS
LIN {X -0.003,Y -507.017,Z 1248.412,A 0.000,B 0.000,C 90.000,E1 290.120} C_DIS
LIN {X -0.150,Y -505.865,Z 1248.397,A 0.000,B 0.000,C 90.000,E1 287.457} C_DIS
LIN {X -0.051,Y -505.568,Z 1248.392,A 0.000,B 0.000,C 90.000,E1 286.551} C_DIS
LIN {X -0.163,Y -505.078,Z 1248.385,A 0.000,B 0.000,C 90.000,E1 285.371} C_DIS
LIN {X -0.209,Y -504.185,Z 1248.377,A 0.000,B 0.000,C 90.000,E1 283.883} C_DIS
LIN {X 0.029,Y -502.940,Z 1248.367,A 0.000,B 0.000,C 90.000,E1 282.063} C_DIS
LIN {X -0.224,Y -502.076,Z 1248.360,A 0.000,B 0.000,C 90.000,E1 280.894} C_DIS
LIN {X 0.202,Y -500.623,Z 1248.349,A 0.000,B 0.000,C 90.000,E1 278.746} C_DIS
LIN {X -0.059,Y -499.107,Z 1248.335,A 0.000,B 0.000,C 90.000,E1 276.372} C_DIS
LIN {X 0.244,Y -498.262,Z 1248.325,A 0.000,B 0.000,C 90.000,E1 274.531} C_DIS
LIN {X 0.128,Y -497.378,Z 1248.317,A 0.000,B 0.000,C 90.000,E1 273.037} C_DIS
LIN {X 0.086,Y -496.517,Z 1248.310,A 0.000,B 0.000,C 90.000,E1 271.835} C_DIS
LIN {X -0.153,Y -494.477,Z 1248.295,A 0.000,B 0.000,C 90.000,E1 269.141} C_DIS
LIN {X -0.019,Y -493.221,Z 1248.285,A 0.000,B 0.000,C 90.000,E1 267.306} C_DIS
LIN {X 0.200,Y -492.874,Z 1248.282,A 0.000,B 0.000,C 90.000,E1 266.674} C_DIS
LIN {X -0.165,Y -491.899,Z 1248.272,A 0.000,B 0.000,C 90.000,E1 264.894} C_DIS
LIN {X -0.066,Y -491.372,Z 1248.266,A 0.000,B 0.000,C 90.000,E1 263.970} C_DIS
LIN {X -0.141,Y -490.501,Z 1248.260,A 0.000,B 0.000,C 90.000,E1 262.761} C_DIS
LIN {X 0.200,Y -489.156,Z 1248.251,A 0.000,B 0.000,C 90.000,E1 261.197} C_DIS
LIN {X 0.033,Y -486.596,Z 1248.236,A 0.000,B 0.000,C 90.000,E1 258.465} C_DIS
LIN {X 0.000,Y -485.477,Z 1248.227,A 0.000,B 0.000,C 90.000,E1 256.937} C_DIS
LIN {X 0.077,Y -484.747,Z 1248.221,A 0.000,B 0.000,C 90.000,E1 255.700} C_DIS
LIN {X -0.016,Y -483.491,Z 1248.209,A 0.000,B 0.000,C 90.000,E1 253.559} C_DIS
LIN {X -0.010,Y -482.256,Z 1248.197,A 0.000,B 0.000,C 90.000,E1 251.402} C_DIS
LIN {X -0.180,Y -481.305,Z 1248.186,A 0.000,B 0.000,C 90.000,E1 249.571} C_DIS
LIN {X 0.256,Y -480.520,Z 1248.178,A 0.000,B 0.000,C 90.000,E1 247.975} C_DIS
LIN {X -0.218,Y -479.621,Z 1248.169,A 0.000,B 0.000,C 90.000,E1 246.485} C_DIS
LIN {X -0.081,Y -478.543,Z 1248.161,A 0.000,B 0.000,C 90.000,E1 244.921} C_DIS
LIN {X -0.005,Y -477.224,Z 1248.150,A 0.000,B 0.000,C 90.000,E1 243.050} C_DIS
LIN {X 0.127,Y -476.610,Z 1248.145,A 0.000,B 0.000,C 90.000,E1 242.103} C_DIS
LIN {X -0.219,Y -475.420,Z 1248.136,A 0.000,B 0.000,C 90.000,E1 240.589} C_DIS
LIN {X 0.248,Y -473.805,Z 1248.126,A 0.000,B 0.000,C 90.000,E1 238.663} C_DIS
LIN {X -0.016,Y -471.293,Z 1248.110,A 0.000,B 0.000,C 90.000,E1 235.881} C_DIS
LIN {X -0.159,Y -469.536,Z 1248.098,A 0.000,B 0.000,C 90.000,E1 233.703} C_DIS
LIN {X 0.216,Y -468.151,Z 1248.086,A 0.000,B 0.000,C 90.000,E1 231.457} C_DIS
LIN {X -0.001,Y -467.175,Z 1248.077,A 0.000,B 0.000,C 90.000,E1 229.908} C_DIS
LIN {X -0.003,Y -466.388,Z 1248.070,A 0.000,B 0.000,C 90.000,E1 228.647} C_DIS
LIN {X -0.186,Y -464.872,Z 1248.058,A 0.000,B 0.000,C 90.000,E1 226.458} C_DIS
LIN {X 0.205,Y -463.091,Z 1248.037,A 0.000,B 0.000,C 90.000,E1 222.609} C_DIS
LIN {X 0.069,Y -464.335,Z 1248.000,A 0.000,B 0.000,C 90.000,E1 215.964} C_DIS
LIN {X 0.028,Y -467.644,Z 1247.975,A 0.000,B 0.000,C 90.000,E1 211.544} C_DIS
LIN {X 0.021,Y -470.367,Z 1247.961,A 0.000,B 0.000,C 90.000,E1 209.027} C_DIS
LIN {X 0.160,Y -472.741,Z 1247.951,A 0.000,B 0.000,C 90.000,E1 207.129} C_DIS
LIN {X 0.005,Y -476.741,Z 1247.934,A 0.000,B 0.000,C 90.000,E1 204.027} C_DIS
LIN {X 0.084,Y -480.083,Z 1247.922,A 0.000,B 0.000,C 90.000,E1 201.844} C_DIS
LIN {X -0.087,Y -485.654,Z 1247.904,A 0.000,B 0.000,C 90.000,E1 198.779} C_DIS
LIN {X 0.131,Y -488.816,Z 1247.896,A 0.000,B 0.000,C 90.000,E1 197.221} C_DIS
LIN {X -0.171,Y -492.871,Z 1247.886,A 0.000,B 0.000,C 90.000,E1 195.426} C_DIS
LIN {X -0.042,Y -497.016,Z 1247.875,A 0.000,B 0.000,C 90.000,E1 193.592} C_DIS
LIN {X -0.144,Y -503.358,Z 1247.860,A 0.000,B 0.000,C 90.000,E1 190.894} C_DIS
LIN {X -0.081,Y -507.829,Z 1247.851,A 0.000,B 0.000,C 90.000,E1 189.095} C_DIS
LIN {X 0.082,Y -512.329,Z 1247.841,A 0.000,B 0.000,C 90.000,E1 187.296} C_DIS
LIN {X 0.218,Y -516.842,Z 1247.831,A 0.000,B 0.000,C 90.000,E1 185.511} C_DIS
LIN {X -0.122,Y -521.936,Z 1247.819,A 0.000,B 0.000,C 90.000,E1 183.498} C_DIS
LIN {X 0.238,Y -524.790,Z 1247.813,A 0.000,B 0.000,C 90.000,E1 182.293} C_DIS
LIN {X 0.086,Y -528.359,Z 1247.805,A 0.000,B 0.000,C 90.000,E1 180.859} C_DIS
LIN {X -0.031,Y -532.489,Z 1247.795,A 0.000,B 0.000,C 90.000,E1 179.141} C_DIS
LIN {X -0.045,Y -535.218,Z 1247.789,A 0.000,B 0.000,C 90.000,E1 177.993} C_DIS
LIN {X -0.008,Y -538.337,Z 1247.781,A 0.000,B 0.000,C 90.000,E1 176.560} C_DIS
LIN {X 0.062,Y -540.742,Z 1247.775,A 0.000,B 0.000,C 90.000,E1 175.412} C_DIS
LIN {X 0.221,Y -543.561,Z 1247.767,A 0.000,B 0.000,C 90.000,E1 173.976} C_DIS
LIN {X 0.033,Y -546.761,Z 1247.757,A 0.000,B 0.000,C 90.000,E1 172.299} C_DIS
LIN {X -0.103,Y -549.219,Z 1247.750,A 0.000,B 0.000,C 90.000,E1 170.905} C_DIS
LIN {X -0.192,Y -551.500,Z 1247.742,A 0.000,B 0.000,C 90.000,E1 169.511} C_DIS
LIN {X 0.282,Y -553.290,Z 1247.735,A 0.000,B 0.000,C 90.000,E1 168.342} C_DIS
LIN {X -0.175,Y -555.452,Z 1247.728,A 0.000,B 0.000,C 90.000,E1 166.992} C_DIS
LIN {X -0.196,Y -557.091,Z 1247.721,A 0.000,B 0.000,C 90.000,E1 165.880} C_DIS
END
